LIN {X 0,Y 566.531,Z 316.319,A -85,B 0,C 180,E1 -2651.108,E2 -2651.108} C_VEL
LIN {X 0,Y 566.471,Z 313.294,A -85,B 0,C 180,E1 -2653.028,E2 -2653.028} C_VEL
LIN {X 0,Y 566.256,Z 311.81,A -85,B 0,C 180,E1 -2654.03,E2 -2654.03} C_VEL
LIN {X 0,Y 566.196,Z 311.46,A -85,B 0,C 180,E1 -2656.049,E2 -2656.049} C_VEL
LIN {X 0,Y 566.205,Z 311.453,A -85,B 0,C 180,E1 -2659.214,E2 -2659.214} C_VEL
LIN {X 0,Y 566.187,Z 311.457,A -85,B 0,C 180,E1 -2661.637,E2 -2661.637} C_VEL
LIN {X 0,Y 566.162,Z 311.463,A -85,B 0,C 180,E1 -2664.308,E2 -2664.308} C_VEL
LIN {X 0,Y 566.22,Z 311.449,A -85,B 0,C 180,E1 -2666.897,E2 -2666.897} C_VEL
LIN {X 0,Y 566.18,Z 311.456,A -85,B 0,C 180,E1 -2669.407,E2 -2669.407} C_VEL
LIN {X 0,Y 566.212,Z 311.46,A -85,B 0,C 180,E1 -2671.857,E2 -2671.857} C_VEL
LIN {X 0,Y 566.214,Z 311.452,A -85,B 0,C 180,E1 -2674.251,E2 -2674.251} C_VEL
LIN {X 0,Y 566.169,Z 311.455,A -85,B 0,C 180,E1 -2676.719,E2 -2676.719} C_VEL
LIN {X 0,Y 566.207,Z 311.46,A -85,B 0,C 180,E1 -2679.662,E2 -2679.662} C_VEL
LIN {X 0,Y 566.198,Z 311.451,A -85,B 0,C 180,E1 -2682.668,E2 -2682.668} C_VEL
LIN {X 0,Y 566.234,Z 311.455,A -85,B 0,C 180,E1 -2685.626,E2 -2685.626} C_VEL
LIN {X 0,Y 566.235,Z 311.447,A -85,B 0,C 180,E1 -2688.675,E2 -2688.675} C_VEL
LIN {X 0,Y 566.233,Z 311.456,A -85,B 0,C 180,E1 -2691.434,E2 -2691.434} C_VEL
LIN {X 0,Y 566.262,Z 311.443,A -85,B 0,C 180,E1 -2694.301,E2 -2694.301} C_VEL
LIN {X 0,Y 566.286,Z 311.442,A -85,B 0,C 180,E1 -2697.866,E2 -2697.866} C_VEL
LIN {X 0,Y 566.297,Z 311.442,A -85,B 0,C 180,E1 -2700.711,E2 -2700.711} C_VEL
LIN {X 0,Y 566.268,Z 311.448,A -85,B 0,C 180,E1 -2702.845,E2 -2702.845} C_VEL
LIN {X 0,Y 566.266,Z 311.444,A -85,B 0,C 180,E1 -2705.698,E2 -2705.698} C_VEL
LIN {X 0,Y 566.226,Z 311.452,A -85,B 0,C 180,E1 -2708.565,E2 -2708.565} C_VEL
LIN {X 0,Y 566.241,Z 311.448,A -85,B 0,C 180,E1 -2711.454,E2 -2711.454} C_VEL
LIN {X 0,Y 566.233,Z 311.452,A -85,B 0,C 180,E1 -2714.506,E2 -2714.506} C_VEL
LIN {X 0,Y 566.197,Z 311.453,A -85,B 0,C 180,E1 -2717.331,E2 -2717.331} C_VEL
LIN {X 0,Y 566.211,Z 311.454,A -85,B 0,C 180,E1 -2720.337,E2 -2720.337} C_VEL
LIN {X 0,Y 566.17,Z 311.456,A -85,B 0,C 180,E1 -2723.281,E2 -2723.281} C_VEL
LIN {X 0,Y 566.212,Z 311.45,A -85,B 0,C 180,E1 -2725.749,E2 -2725.749} C_VEL
LIN {X 0,Y 566.201,Z 311.451,A -85,B 0,C 180,E1 -2727.472,E2 -2727.472} C_VEL
LIN {X 0,Y 565.52,Z 311.541,A -85,B 0,C 180,E1 -2728.066,E2 -2728.066} C_VEL
LIN {X 0,Y 562.655,Z 311.896,A -85,B 0,C 180,E1 -2729.029,E2 -2729.029} C_VEL
LIN {X 0,Y 560.247,Z 312.196,A -85,B 0,C 180,E1 -2729.805,E2 -2729.805} C_VEL
LIN {X 0,Y 559.222,Z 312.33,A -85,B 0,C 180,E1 -2730.404,E2 -2730.404} C_VEL
LIN {X 0,Y 559.142,Z 312.332,A -85,B 0,C 180,E1 -2730.606,E2 -2730.606} C_VEL
LIN {X 0,Y 559.173,Z 312.331,A -85,B 0,C 180,E1 -2732.714,E2 -2732.714} C_VEL
LIN {X 0,Y 559.141,Z 312.33,A -85,B 0,C 180,E1 -2735.323,E2 -2735.323} C_VEL
LIN {X 0,Y 559.133,Z 312.337,A -85,B 0,C 180,E1 -2738.017,E2 -2738.017} C_VEL
LIN {X 0,Y 559.173,Z 312.328,A -85,B 0,C 180,E1 -2740.81,E2 -2740.81} C_VEL
LIN {X 0,Y 559.16,Z 312.332,A -85,B 0,C 180,E1 -2743.731,E2 -2743.731} C_VEL
LIN {X 0,Y 559.146,Z 312.33,A -85,B 0,C 180,E1 -2746.803,E2 -2746.803} C_VEL
LIN {X 0,Y 559.173,Z 312.327,A -85,B 0,C 180,E1 -2749.189,E2 -2749.189} C_VEL
LIN {X 0,Y 559.132,Z 312.34,A -85,B 0,C 180,E1 -2751.983,E2 -2751.983} C_VEL
LIN {X 0,Y 559.143,Z 312.33,A -85,B 0,C 180,E1 -2754.785,E2 -2754.785} C_VEL
LIN {X 0,Y 559.171,Z 312.33,A -85,B 0,C 180,E1 -2757.361,E2 -2757.361} C_VEL
LIN {X 0,Y 559.146,Z 312.333,A -85,B 0,C 180,E1 -2760.142,E2 -2760.142} C_VEL
LIN {X 0,Y 559.179,Z 312.328,A -85,B 0,C 180,E1 -2763.17,E2 -2763.17} C_VEL
LIN {X 0,Y 559.154,Z 312.337,A -85,B 0,C 180,E1 -2765.495,E2 -2765.495} C_VEL
LIN {X 0,Y 559.169,Z 312.327,A -85,B 0,C 180,E1 -2768.624,E2 -2768.624} C_VEL
LIN {X 0,Y 559.166,Z 312.33,A -85,B 0,C 180,E1 -2770.926,E2 -2770.926} C_VEL
LIN {X 0,Y 559.164,Z 312.331,A -85,B 0,C 180,E1 -2773.948,E2 -2773.948} C_VEL
LIN {X 0,Y 559.169,Z 312.328,A -85,B 0,C 180,E1 -2776.184,E2 -2776.184} C_VEL
LIN {X 0,Y 559.194,Z 312.332,A -85,B 0,C 180,E1 -2779.134,E2 -2779.134} C_VEL
LIN {X 0,Y 559.203,Z 312.324,A -85,B 0,C 180,E1 -2782.054,E2 -2782.054} C_VEL
LIN {X 0,Y 559.253,Z 312.325,A -85,B 0,C 180,E1 -2784.953,E2 -2784.953} C_VEL
LIN {X 0,Y 559.255,Z 312.318,A -85,B 0,C 180,E1 -2787.839,E2 -2787.839} C_VEL
LIN {X 0,Y 559.27,Z 312.321,A -85,B 0,C 180,E1 -2790.72,E2 -2790.72} C_VEL
LIN {X 0,Y 559.236,Z 312.328,A -85,B 0,C 180,E1 -2792.881,E2 -2792.881} C_VEL
LIN {X 0,Y 559.235,Z 312.32,A -85,B 0,C 180,E1 -2795.77,E2 -2795.77} C_VEL
LIN {X 0,Y 559.189,Z 312.333,A -85,B 0,C 180,E1 -2798.674,E2 -2798.674} C_VEL
LIN {X 0,Y 559.202,Z 312.324,A -85,B 0,C 180,E1 -2801.6,E2 -2801.6} C_VEL
LIN {X 0,Y 559.197,Z 312.333,A -85,B 0,C 180,E1 -2804.596,E2 -2804.596} C_VEL
LIN {X 0,Y 559.157,Z 312.33,A -85,B 0,C 180,E1 -2807.557,E2 -2807.557} C_VEL
LIN {X 0,Y 559.17,Z 312.328,A -85,B 0,C 180,E1 -2809.837,E2 -2809.837} C_VEL
LIN {X 0,Y 559.139,Z 312.336,A -85,B 0,C 180,E1 -2812.153,E2 -2812.153} C_VEL
LIN {X 0,Y 559.175,Z 312.326,A -85,B 0,C 180,E1 -2815.298,E2 -2815.298} C_VEL
LIN {X 0,Y 559.192,Z 312.326,A -85,B 0,C 180,E1 -2817.711,E2 -2817.711} C_VEL
LIN {X 0,Y 559.16,Z 312.329,A -85,B 0,C 180,E1 -2821.019,E2 -2821.019} C_VEL
LIN {X 0,Y 559.162,Z 312.334,A -85,B 0,C 180,E1 -2823.949,E2 -2823.949} C_VEL
LIN {X 0,Y 559.142,Z 312.33,A -85,B 0,C 180,E1 -2827.108,E2 -2827.108} C_VEL
LIN {X 0,Y 559.167,Z 312.336,A -85,B 0,C 180,E1 -2829.943,E2 -2829.943} C_VEL
LIN {X 0,Y 559.16,Z 312.329,A -85,B 0,C 180,E1 -2832.743,E2 -2832.743} C_VEL
LIN {X 0,Y 559.152,Z 312.337,A -85,B 0,C 180,E1 -2835.761,E2 -2835.761} C_VEL
LIN {X 0,Y 559.189,Z 312.328,A -85,B 0,C 180,E1 -2838.233,E2 -2838.233} C_VEL
LIN {X 0,Y 559.175,Z 312.328,A -85,B 0,C 180,E1 -2841.191,E2 -2841.191} C_VEL
LIN {X 0,Y 559.136,Z 312.339,A -85,B 0,C 180,E1 -2843.79,E2 -2843.79} C_VEL
LIN {X 0,Y 559.162,Z 312.328,A -85,B 0,C 180,E1 -2846.426,E2 -2846.426} C_VEL
LIN {X 0,Y 559.16,Z 312.33,A -85,B 0,C 180,E1 -2848.982,E2 -2848.982} C_VEL
LIN {X 0,Y 559.165,Z 312.335,A -85,B 0,C 180,E1 -2851.619,E2 -2851.619} C_VEL
LIN {X 0,Y 559.179,Z 312.329,A -85,B 0,C 180,E1 -2853.903,E2 -2853.903} C_VEL
LIN {X 0,Y 559.14,Z 312.331,A -85,B 0,C 180,E1 -2856.571,E2 -2856.571} C_VEL
LIN {X 0,Y 559.178,Z 312.335,A -85,B 0,C 180,E1 -2859.396,E2 -2859.396} C_VEL
LIN {X 0,Y 559.144,Z 312.333,A -85,B 0,C 180,E1 -2861.686,E2 -2861.686} C_VEL
LIN {X 0,Y 559.163,Z 312.328,A -85,B 0,C 180,E1 -2863.948,E2 -2863.948} C_VEL
LIN {X 0,Y 559.17,Z 312.327,A -85,B 0,C 180,E1 -2866.184,E2 -2866.184} C_VEL
LIN {X 0,Y 559.194,Z 312.333,A -85,B 0,C 180,E1 -2869.134,E2 -2869.134} C_VEL
LIN {X 0,Y 559.202,Z 312.323,A -85,B 0,C 180,E1 -2872.054,E2 -2872.054} C_VEL
LIN {X 0,Y 559.252,Z 312.327,A -85,B 0,C 180,E1 -2874.954,E2 -2874.954} C_VEL
LIN {X 0,Y 559.255,Z 312.316,A -85,B 0,C 180,E1 -2877.84,E2 -2877.84} C_VEL
LIN {X 0,Y 559.274,Z 312.322,A -85,B 0,C 180,E1 -2880.72,E2 -2880.72} C_VEL
LIN {X 0,Y 559.237,Z 312.326,A -85,B 0,C 180,E1 -2882.882,E2 -2882.882} C_VEL
LIN {X 0,Y 559.231,Z 312.319,A -85,B 0,C 180,E1 -2885.771,E2 -2885.771} C_VEL
LIN {X 0,Y 559.191,Z 312.333,A -85,B 0,C 180,E1 -2888.675,E2 -2888.675} C_VEL
LIN {X 0,Y 559.205,Z 312.323,A -85,B 0,C 180,E1 -2891.601,E2 -2891.601} C_VEL
LIN {X 0,Y 559.2,Z 312.331,A -85,B 0,C 180,E1 -2894.596,E2 -2894.596} C_VEL
LIN {X 0,Y 559.142,Z 312.331,A -85,B 0,C 180,E1 -2897.558,E2 -2897.558} C_VEL
LIN {X 0,Y 559.166,Z 312.33,A -85,B 0,C 180,E1 -2899.838,E2 -2899.838} C_VEL
LIN {X 0,Y 559.142,Z 312.338,A -85,B 0,C 180,E1 -2902.153,E2 -2902.153} C_VEL
LIN {X 0,Y 559.176,Z 312.326,A -85,B 0,C 180,E1 -2905.298,E2 -2905.298} C_VEL
LIN {X 0,Y 559.157,Z 312.332,A -85,B 0,C 180,E1 -2907.714,E2 -2907.714} C_VEL
LIN {X 0,Y 559.153,Z 312.337,A -85,B 0,C 180,E1 -2910.183,E2 -2910.183} C_VEL
LIN {X 0,Y 559.157,Z 312.329,A -85,B 0,C 180,E1 -2912.716,E2 -2912.716} C_VEL
LIN {X 0,Y 559.127,Z 312.333,A -85,B 0,C 180,E1 -2915.324,E2 -2915.324} C_VEL
LIN {X 0,Y 559.134,Z 312.341,A -85,B 0,C 180,E1 -2918.018,E2 -2918.018} C_VEL
LIN {X 0,Y 559.156,Z 312.331,A -85,B 0,C 180,E1 -2920.813,E2 -2920.813} C_VEL
LIN {X 0,Y 559.14,Z 312.34,A -85,B 0,C 180,E1 -2923.734,E2 -2923.734} C_VEL
LIN {X 0,Y 559.151,Z 312.338,A -85,B 0,C 180,E1 -2925.262,E2 -2925.262} C_VEL
LIN {X 0,Y 559.431,Z 314.242,A -85,B 0,C 180,E1 -2926.773,E2 -2926.773} C_VEL
LIN {X 0,Y 559.539,Z 318.057,A -85,B 0,C 180,E1 -2929.222,E2 -2929.222} C_VEL
LIN {X 0,Y 559.468,Z 322.75,A -85,B 0,C 180,E1 -2932.009,E2 -2932.009} C_VEL
LIN {X 0,Y 559.387,Z 327.696,A -85,B 0,C 180,E1 -2934.751,E2 -2934.751} C_VEL
LIN {X 0,Y 559.313,Z 332.663,A -85,B 0,C 180,E1 -2937.34,E2 -2937.34} C_VEL
LIN {X 0,Y 559.203,Z 338.301,A -85,B 0,C 180,E1 -2940.134,E2 -2940.134} C_VEL
LIN {X 0,Y 559.094,Z 344.792,A -85,B 0,C 180,E1 -2943.189,E2 -2943.189} C_VEL
LIN {X 0,Y 559.019,Z 349.846,A -85,B 0,C 180,E1 -2945.489,E2 -2945.489} C_VEL
LIN {X 0,Y 558.987,Z 357.018,A -85,B 0,C 180,E1 -2948.617,E2 -2948.617} C_VEL
LIN {X 0,Y 558.928,Z 362.478,A -85,B 0,C 180,E1 -2950.918,E2 -2950.918} C_VEL
LIN {X 0,Y 558.876,Z 367.867,A -85,B 0,C 180,E1 -2953.188,E2 -2953.188} C_VEL
LIN {X 0,Y 558.841,Z 375.053,A -85,B 0,C 180,E1 -2956.176,E2 -2956.176} C_VEL
LIN {X 0,Y 558.832,Z 377.523,A -85,B 0,C 180,E1 -2957.194,E2 -2957.194} C_VEL
LIN {X 0,Y 559.957,Z 385.372,A -85,B 0,C 180,E1 -2957.381,E2 -2957.381} C_VEL
LIN {X 0,Y 559.843,Z 397.181,A -85,B 0,C 180,E1 -2957.728,E2 -2957.728} C_VEL
LIN {X 0,Y 559.719,Z 408.183,A -85,B 0,C 180,E1 -2958.171,E2 -2958.171} C_VEL
LIN {X 0,Y 559.565,Z 418.532,A -85,B 0,C 180,E1 -2958.704,E2 -2958.704} C_VEL
LIN {X 0,Y 559.421,Z 429.49,A -85,B 0,C 180,E1 -2959.413,E2 -2959.413} C_VEL
LIN {X 0,Y 559.289,Z 439.624,A -85,B 0,C 180,E1 -2960.233,E2 -2960.233} C_VEL
LIN {X 0,Y 559.138,Z 448.736,A -85,B 0,C 180,E1 -2961.143,E2 -2961.143} C_VEL
LIN {X 0,Y 559.052,Z 456.283,A -85,B 0,C 180,E1 -2962.051,E2 -2962.051} C_VEL
LIN {X 0,Y 558.934,Z 462.688,A -85,B 0,C 180,E1 -2962.976,E2 -2962.976} C_VEL
LIN {X 0,Y 558.908,Z 467.807,A -85,B 0,C 180,E1 -2963.864,E2 -2963.864} C_VEL
LIN {X 0,Y 558.798,Z 472.904,A -85,B 0,C 180,E1 -2964.949,E2 -2964.949} C_VEL
LIN {X 0,Y 558.844,Z 476.858,A -85,B 0,C 180,E1 -2966.034,E2 -2966.034} C_VEL
LIN {X 0,Y 558.799,Z 479.778,A -85,B 0,C 180,E1 -2967.116,E2 -2967.116} C_VEL
LIN {X 0,Y 558.745,Z 482.194,A -85,B 0,C 180,E1 -2968.559,E2 -2968.559} C_VEL
LIN {X 0,Y 558.741,Z 482.781,A -85,B 0,C 180,E1 -2969.279,E2 -2969.279} C_VEL
LIN {X 0,Y 558.741,Z 482.781,A -85,B 0,C 180,E1 -2970.721,E2 -2970.721} C_VEL
LIN {X 0,Y 558.745,Z 482.194,A -85,B 0,C 180,E1 -2971.441,E2 -2971.441} C_VEL
LIN {X 0,Y 558.799,Z 479.778,A -85,B 0,C 180,E1 -2972.884,E2 -2972.884} C_VEL
LIN {X 0,Y 558.844,Z 476.858,A -85,B 0,C 180,E1 -2973.966,E2 -2973.966} C_VEL
LIN {X 0,Y 558.798,Z 472.904,A -85,B 0,C 180,E1 -2975.051,E2 -2975.051} C_VEL
LIN {X 0,Y 558.91,Z 467.807,A -85,B 0,C 180,E1 -2976.136,E2 -2976.136} C_VEL
LIN {X 0,Y 558.975,Z 461.423,A -85,B 0,C 180,E1 -2977.223,E2 -2977.223} C_VEL
LIN {X 0,Y 559.093,Z 453.5,A -85,B 0,C 180,E1 -2978.312,E2 -2978.312} C_VEL
LIN {X 0,Y 559.21,Z 445.358,A -85,B 0,C 180,E1 -2979.221,E2 -2979.221} C_VEL
LIN {X 0,Y 559.345,Z 435.315,A -85,B 0,C 180,E1 -2980.131,E2 -2980.131} C_VEL
LIN {X 0,Y 559.473,Z 426.835,A -85,B 0,C 180,E1 -2980.769,E2 -2980.769} C_VEL
LIN {X 0,Y 559.575,Z 416.58,A -85,B 0,C 180,E1 -2981.405,E2 -2981.405} C_VEL
LIN {X 0,Y 559.736,Z 405.396,A -85,B 0,C 180,E1 -2981.956,E2 -2981.956} C_VEL
LIN {X 0,Y 559.931,Z 392.286,A -85,B 0,C 180,E1 -2982.435,E2 -2982.435} C_VEL
LIN {X 0,Y 559.761,Z 383.139,A -85,B 0,C 180,E1 -2982.678,E2 -2982.678} C_VEL
LIN {X 0,Y 558.832,Z 377.523,A -85,B 0,C 180,E1 -2982.806,E2 -2982.806} C_VEL
LIN {X 0,Y 558.852,Z 371.46,A -85,B 0,C 180,E1 -2985.313,E2 -2985.313} C_VEL
LIN {X 0,Y 558.903,Z 364.274,A -85,B 0,C 180,E1 -2988.322,E2 -2988.322} C_VEL
LIN {X 0,Y 558.932,Z 358.847,A -85,B 0,C 180,E1 -2990.614,E2 -2990.614} C_VEL
LIN {X 0,Y 558.97,Z 352.352,A -85,B 0,C 180,E1 -2993.387,E2 -2993.387} C_VEL
LIN {X 0,Y 559.064,Z 346.339,A -85,B 0,C 180,E1 -2996.103,E2 -2996.103} C_VEL
LIN {X 0,Y 559.116,Z 341.086,A -85,B 0,C 180,E1 -2998.532,E2 -2998.532} C_VEL
LIN {X 0,Y 559.232,Z 335.376,A -85,B 0,C 180,E1 -3001.287,E2 -3001.287} C_VEL
LIN {X 0,Y 559.298,Z 330.113,A -85,B 0,C 180,E1 -3003.969,E2 -3003.969} C_VEL
LIN {X 0,Y 559.418,Z 325.417,A -85,B 0,C 180,E1 -3006.482,E2 -3006.482} C_VEL
LIN {X 0,Y 559.507,Z 321.151,A -85,B 0,C 180,E1 -3008.906,E2 -3008.906} C_VEL
LIN {X 0,Y 559.54,Z 316.507,A -85,B 0,C 180,E1 -3011.736,E2 -3011.736} C_VEL
LIN {X 0,Y 559.319,Z 313.521,A -85,B 0,C 180,E1 -3013.716,E2 -3013.716} C_VEL
LIN {X 0,Y 559.151,Z 312.337,A -85,B 0,C 180,E1 -3014.738,E2 -3014.738} C_VEL
LIN {X 0,Y 559.156,Z 312.336,A -85,B 0,C 180,E1 -3017.865,E2 -3017.865} C_VEL
LIN {X 0,Y 559.185,Z 312.335,A -85,B 0,C 180,E1 -3020.134,E2 -3020.134} C_VEL
LIN {X 0,Y 559.141,Z 312.332,A -85,B 0,C 180,E1 -3022.891,E2 -3022.891} C_VEL
LIN {X 0,Y 559.166,Z 312.336,A -85,B 0,C 180,E1 -3026.051,E2 -3026.051} C_VEL
LIN {X 0,Y 559.155,Z 312.329,A -85,B 0,C 180,E1 -3028.98,E2 -3028.98} C_VEL
LIN {X 0,Y 559.169,Z 312.333,A -85,B 0,C 180,E1 -3031.618,E2 -3031.618} C_VEL
LIN {X 0,Y 559.18,Z 312.334,A -85,B 0,C 180,E1 -3033.903,E2 -3033.903} C_VEL
LIN {X 0,Y 559.139,Z 312.331,A -85,B 0,C 180,E1 -3036.571,E2 -3036.571} C_VEL
LIN {X 0,Y 559.176,Z 312.331,A -85,B 0,C 180,E1 -3039.395,E2 -3039.395} C_VEL
LIN {X 0,Y 559.142,Z 312.339,A -85,B 0,C 180,E1 -3041.685,E2 -3041.685} C_VEL
LIN {X 0,Y 559.166,Z 312.331,A -85,B 0,C 180,E1 -3043.947,E2 -3043.947} C_VEL
LIN {X 0,Y 559.17,Z 312.328,A -85,B 0,C 180,E1 -3046.184,E2 -3046.184} C_VEL
LIN {X 0,Y 559.196,Z 312.328,A -85,B 0,C 180,E1 -3049.133,E2 -3049.133} C_VEL
LIN {X 0,Y 559.201,Z 312.324,A -85,B 0,C 180,E1 -3052.053,E2 -3052.053} C_VEL
LIN {X 0,Y 559.254,Z 312.321,A -85,B 0,C 180,E1 -3054.953,E2 -3054.953} C_VEL
LIN {X 0,Y 559.256,Z 312.318,A -85,B 0,C 180,E1 -3057.839,E2 -3057.839} C_VEL
LIN {X 0,Y 559.268,Z 312.318,A -85,B 0,C 180,E1 -3060.72,E2 -3060.72} C_VEL
LIN {X 0,Y 559.235,Z 312.325,A -85,B 0,C 180,E1 -3062.881,E2 -3062.881} C_VEL
LIN {X 0,Y 559.234,Z 312.32,A -85,B 0,C 180,E1 -3065.77,E2 -3065.77} C_VEL
LIN {X 0,Y 559.185,Z 312.33,A -85,B 0,C 180,E1 -3068.674,E2 -3068.674} C_VEL
LIN {X 0,Y 559.204,Z 312.324,A -85,B 0,C 180,E1 -3071.6,E2 -3071.6} C_VEL
LIN {X 0,Y 559.198,Z 312.329,A -85,B 0,C 180,E1 -3074.595,E2 -3074.595} C_VEL
LIN {X 0,Y 559.157,Z 312.329,A -85,B 0,C 180,E1 -3077.557,E2 -3077.557} C_VEL
LIN {X 0,Y 559.17,Z 312.327,A -85,B 0,C 180,E1 -3079.837,E2 -3079.837} C_VEL
LIN {X 0,Y 559.14,Z 312.333,A -85,B 0,C 180,E1 -3082.152,E2 -3082.152} C_VEL
LIN {X 0,Y 559.173,Z 312.327,A -85,B 0,C 180,E1 -3085.298,E2 -3085.298} C_VEL
LIN {X 0,Y 559.178,Z 312.326,A -85,B 0,C 180,E1 -3087.712,E2 -3087.712} C_VEL
LIN {X 0,Y 559.142,Z 312.332,A -85,B 0,C 180,E1 -3090.606,E2 -3090.606} C_VEL
LIN {X 0,Y 558.482,Z 312.415,A -85,B 0,C 180,E1 -3091.208,E2 -3091.208} C_VEL
LIN {X 0,Y 555.622,Z 312.775,A -85,B 0,C 180,E1 -3092.184,E2 -3092.184} C_VEL
LIN {X 0,Y 553.208,Z 313.072,A -85,B 0,C 180,E1 -3092.97,E2 -3092.97} C_VEL
LIN {X 0,Y 552.185,Z 313.198,A -85,B 0,C 180,E1 -3093.576,E2 -3093.576} C_VEL
LIN {X 0,Y 552.11,Z 313.208,A -85,B 0,C 180,E1 -3093.782,E2 -3093.782} C_VEL
LIN {X 0,Y 552.106,Z 313.21,A -85,B 0,C 180,E1 -3096.746,E2 -3096.746} C_VEL
LIN {X 0,Y 552.131,Z 313.205,A -85,B 0,C 180,E1 -3099.526,E2 -3099.526} C_VEL
LIN {X 0,Y 552.127,Z 313.209,A -85,B 0,C 180,E1 -3102.425,E2 -3102.425} C_VEL
LIN {X 0,Y 552.096,Z 313.21,A -85,B 0,C 180,E1 -3105.563,E2 -3105.563} C_VEL
LIN {X 0,Y 552.137,Z 313.204,A -85,B 0,C 180,E1 -3108.676,E2 -3108.676} C_VEL
LIN {X 0,Y 552.117,Z 313.208,A -85,B 0,C 180,E1 -3111.411,E2 -3111.411} C_VEL
LIN {X 0,Y 552.099,Z 313.213,A -85,B 0,C 180,E1 -3114.158,E2 -3114.158} C_VEL
LIN {X 0,Y 552.12,Z 313.205,A -85,B 0,C 180,E1 -3116.815,E2 -3116.815} C_VEL
LIN {X 0,Y 552.104,Z 313.211,A -85,B 0,C 180,E1 -3119.391,E2 -3119.391} C_VEL
LIN {X 0,Y 552.124,Z 313.211,A -85,B 0,C 180,E1 -3121.903,E2 -3121.903} C_VEL
LIN {X 0,Y 552.154,Z 313.201,A -85,B 0,C 180,E1 -3124.649,E2 -3124.649} C_VEL
LIN {X 0,Y 552.09,Z 313.219,A -85,B 0,C 180,E1 -3127.549,E2 -3127.549} C_VEL
LIN {X 0,Y 552.146,Z 313.202,A -85,B 0,C 180,E1 -3130.373,E2 -3130.373} C_VEL
LIN {X 0,Y 552.152,Z 313.205,A -85,B 0,C 180,E1 -3132.977,E2 -3132.977} C_VEL
LIN {X 0,Y 552.133,Z 313.206,A -85,B 0,C 180,E1 -3136.004,E2 -3136.004} C_VEL
LIN {X 0,Y 552.161,Z 313.206,A -85,B 0,C 180,E1 -3138.993,E2 -3138.993} C_VEL
LIN {X 0,Y 552.157,Z 313.203,A -85,B 0,C 180,E1 -3141.952,E2 -3141.952} C_VEL
LIN {X 0,Y 552.228,Z 313.199,A -85,B 0,C 180,E1 -3144.889,E2 -3144.889} C_VEL
LIN {X 0,Y 552.225,Z 313.194,A -85,B 0,C 180,E1 -3147.812,E2 -3147.812} C_VEL
LIN {X 0,Y 552.24,Z 313.197,A -85,B 0,C 180,E1 -3150.729,E2 -3150.729} C_VEL
LIN {X 0,Y 552.202,Z 313.204,A -85,B 0,C 180,E1 -3152.918,E2 -3152.918} C_VEL
LIN {X 0,Y 552.205,Z 313.196,A -85,B 0,C 180,E1 -3155.844,E2 -3155.844} C_VEL
LIN {X 0,Y 552.16,Z 313.21,A -85,B 0,C 180,E1 -3158.786,E2 -3158.786} C_VEL
LIN {X 0,Y 552.16,Z 313.201,A -85,B 0,C 180,E1 -3161.75,E2 -3161.75} C_VEL
LIN {X 0,Y 552.133,Z 313.213,A -85,B 0,C 180,E1 -3164.748,E2 -3164.748} C_VEL
LIN {X 0,Y 552.108,Z 313.208,A -85,B 0,C 180,E1 -3167.788,E2 -3167.788} C_VEL
LIN {X 0,Y 552.128,Z 313.208,A -85,B 0,C 180,E1 -3170.101,E2 -3170.101} C_VEL
LIN {X 0,Y 552.09,Z 313.219,A -85,B 0,C 180,E1 -3172.451,E2 -3172.451} C_VEL
LIN {X 0,Y 552.154,Z 313.201,A -85,B 0,C 180,E1 -3175.351,E2 -3175.351} C_VEL
LIN {X 0,Y 552.124,Z 313.211,A -85,B 0,C 180,E1 -3178.097,E2 -3178.097} C_VEL
LIN {X 0,Y 552.104,Z 313.211,A -85,B 0,C 180,E1 -3180.609,E2 -3180.609} C_VEL
LIN {X 0,Y 552.12,Z 313.205,A -85,B 0,C 180,E1 -3183.185,E2 -3183.185} C_VEL
LIN {X 0,Y 552.099,Z 313.213,A -85,B 0,C 180,E1 -3185.842,E2 -3185.842} C_VEL
LIN {X 0,Y 552.123,Z 313.205,A -85,B 0,C 180,E1 -3189.062,E2 -3189.062} C_VEL
LIN {X 0,Y 552.137,Z 313.205,A -85,B 0,C 180,E1 -3191.444,E2 -3191.444} C_VEL
LIN {X 0,Y 552.093,Z 313.21,A -85,B 0,C 180,E1 -3194.532,E2 -3194.532} C_VEL
LIN {X 0,Y 552.128,Z 313.21,A -85,B 0,C 180,E1 -3197.585,E2 -3197.585} C_VEL
LIN {X 0,Y 552.131,Z 313.205,A -85,B 0,C 180,E1 -3200.474,E2 -3200.474} C_VEL
LIN {X 0,Y 552.103,Z 313.211,A -85,B 0,C 180,E1 -3203.317,E2 -3203.317} C_VEL
LIN {X 0,Y 552.124,Z 313.21,A -85,B 0,C 180,E1 -3205.939,E2 -3205.939} C_VEL
LIN {X 0,Y 552.116,Z 313.206,A -85,B 0,C 180,E1 -3208.541,E2 -3208.541} C_VEL
LIN {X 0,Y 552.122,Z 313.213,A -85,B 0,C 180,E1 -3211.438,E2 -3211.438} C_VEL
LIN {X 0,Y 552.128,Z 313.204,A -85,B 0,C 180,E1 -3214.356,E2 -3214.356} C_VEL
LIN {X 0,Y 552.097,Z 313.209,A -85,B 0,C 180,E1 -3216.758,E2 -3216.758} C_VEL
LIN {X 0,Y 552.119,Z 313.212,A -85,B 0,C 180,E1 -3219.12,E2 -3219.12} C_VEL
LIN {X 0,Y 552.123,Z 313.211,A -85,B 0,C 180,E1 -3221.445,E2 -3221.445} C_VEL
LIN {X 0,Y 552.113,Z 313.208,A -85,B 0,C 180,E1 -3223.738,E2 -3223.738} C_VEL
LIN {X 0,Y 552.134,Z 313.204,A -85,B 0,C 180,E1 -3226.005,E2 -3226.005} C_VEL
LIN {X 0,Y 552.161,Z 313.208,A -85,B 0,C 180,E1 -3228.994,E2 -3228.994} C_VEL
LIN {X 0,Y 552.156,Z 313.201,A -85,B 0,C 180,E1 -3231.952,E2 -3231.952} C_VEL
LIN {X 0,Y 552.227,Z 313.201,A -85,B 0,C 180,E1 -3234.889,E2 -3234.889} C_VEL
LIN {X 0,Y 552.226,Z 313.192,A -85,B 0,C 180,E1 -3237.812,E2 -3237.812} C_VEL
LIN {X 0,Y 552.244,Z 313.198,A -85,B 0,C 180,E1 -3240.73,E2 -3240.73} C_VEL
LIN {X 0,Y 552.203,Z 313.202,A -85,B 0,C 180,E1 -3242.919,E2 -3242.919} C_VEL
LIN {X 0,Y 552.201,Z 313.195,A -85,B 0,C 180,E1 -3245.844,E2 -3245.844} C_VEL
LIN {X 0,Y 552.162,Z 313.207,A -85,B 0,C 180,E1 -3248.786,E2 -3248.786} C_VEL
LIN {X 0,Y 552.162,Z 313.2,A -85,B 0,C 180,E1 -3251.751,E2 -3251.751} C_VEL
LIN {X 0,Y 552.136,Z 313.208,A -85,B 0,C 180,E1 -3254.749,E2 -3254.749} C_VEL
LIN {X 0,Y 552.1,Z 313.209,A -85,B 0,C 180,E1 -3257.789,E2 -3257.789} C_VEL
LIN {X 0,Y 552.127,Z 313.21,A -85,B 0,C 180,E1 -3260.102,E2 -3260.102} C_VEL
LIN {X 0,Y 552.092,Z 313.215,A -85,B 0,C 180,E1 -3262.451,E2 -3262.451} C_VEL
LIN {X 0,Y 552.156,Z 313.201,A -85,B 0,C 180,E1 -3265.351,E2 -3265.351} C_VEL
LIN {X 0,Y 552.11,Z 313.215,A -85,B 0,C 180,E1 -3268.099,E2 -3268.099} C_VEL
LIN {X 0,Y 552.102,Z 313.21,A -85,B 0,C 180,E1 -3270.61,E2 -3270.61} C_VEL
LIN {X 0,Y 552.116,Z 313.206,A -85,B 0,C 180,E1 -3273.186,E2 -3273.186} C_VEL
LIN {X 0,Y 552.086,Z 313.217,A -85,B 0,C 180,E1 -3275.844,E2 -3275.844} C_VEL
LIN {X 0,Y 552.125,Z 313.207,A -85,B 0,C 180,E1 -3279.062,E2 -3279.062} C_VEL
LIN {X 0,Y 552.122,Z 313.212,A -85,B 0,C 180,E1 -3281.446,E2 -3281.446} C_VEL
LIN {X 0,Y 552.095,Z 313.215,A -85,B 0,C 180,E1 -3284.532,E2 -3284.532} C_VEL
LIN {X 0,Y 552.171,Z 313.752,A -85,B 0,C 180,E1 -3285.57,E2 -3285.57} C_VEL
LIN {X 0,Y 552.532,Z 316.734,A -85,B 0,C 180,E1 -3287.613,E2 -3287.613} C_VEL
LIN {X 0,Y 552.491,Z 321.334,A -85,B 0,C 180,E1 -3290.504,E2 -3290.504} C_VEL
LIN {X 0,Y 552.436,Z 326.103,A -85,B 0,C 180,E1 -3293.279,E2 -3293.279} C_VEL
LIN {X 0,Y 552.298,Z 330.997,A -85,B 0,C 180,E1 -3295.951,E2 -3295.951} C_VEL
LIN {X 0,Y 552.203,Z 336.005,A -85,B 0,C 180,E1 -3298.546,E2 -3298.546} C_VEL
LIN {X 0,Y 552.084,Z 341.909,A -85,B 0,C 180,E1 -3301.446,E2 -3301.446} C_VEL
LIN {X 0,Y 551.994,Z 348.09,A -85,B 0,C 180,E1 -3304.349,E2 -3304.349} C_VEL
LIN {X 0,Y 551.88,Z 355.104,A -85,B 0,C 180,E1 -3307.54,E2 -3307.54} C_VEL
LIN {X 0,Y 551.884,Z 361.908,A -85,B 0,C 180,E1 -3310.452,E2 -3310.452} C_VEL
LIN {X 0,Y 551.816,Z 367.867,A -85,B 0,C 180,E1 -3312.967,E2 -3312.967} C_VEL
LIN {X 0,Y 551.755,Z 375.053,A -85,B 0,C 180,E1 -3315.995,E2 -3315.995} C_VEL
LIN {X 0,Y 551.73,Z 377.523,A -85,B 0,C 180,E1 -3317.026,E2 -3317.026} C_VEL
LIN {X 0,Y 553.023,Z 386.217,A -85,B 0,C 180,E1 -3317.244,E2 -3317.244} C_VEL
LIN {X 0,Y 552.921,Z 397.035,A -85,B 0,C 180,E1 -3317.568,E2 -3317.568} C_VEL
LIN {X 0,Y 552.772,Z 407.382,A -85,B 0,C 180,E1 -3317.984,E2 -3317.984} C_VEL
LIN {X 0,Y 552.622,Z 417.171,A -85,B 0,C 180,E1 -3318.484,E2 -3318.484} C_VEL
LIN {X 0,Y 552.486,Z 426.82,A -85,B 0,C 180,E1 -3319.093,E2 -3319.093} C_VEL
LIN {X 0,Y 552.327,Z 436.435,A -85,B 0,C 180,E1 -3319.831,E2 -3319.831} C_VEL
LIN {X 0,Y 552.153,Z 447.105,A -85,B 0,C 180,E1 -3320.845,E2 -3320.845} C_VEL
LIN {X 0,Y 552.01,Z 454.905,A -85,B 0,C 180,E1 -3321.765,E2 -3321.765} C_VEL
LIN {X 0,Y 551.904,Z 461.415,A -85,B 0,C 180,E1 -3322.684,E2 -3322.684} C_VEL
LIN {X 0,Y 551.809,Z 467.105,A -85,B 0,C 180,E1 -3323.651,E2 -3323.651} C_VEL
LIN {X 0,Y 551.802,Z 471.352,A -85,B 0,C 180,E1 -3324.519,E2 -3324.519} C_VEL
LIN {X 0,Y 551.767,Z 475.643,A -85,B 0,C 180,E1 -3325.617,E2 -3325.617} C_VEL
LIN {X 0,Y 551.75,Z 477.975,A -85,B 0,C 180,E1 -3326.348,E2 -3326.348} C_VEL
LIN {X 0,Y 551.723,Z 479.773,A -85,B 0,C 180,E1 -3327.079,E2 -3327.079} C_VEL
LIN {X 0,Y 551.645,Z 482.196,A -85,B 0,C 180,E1 -3328.54,E2 -3328.54} C_VEL
LIN {X 0,Y 551.641,Z 482.78,A -85,B 0,C 180,E1 -3329.27,E2 -3329.27} C_VEL
LIN {X 0,Y 551.641,Z 482.78,A -85,B 0,C 180,E1 -3330.73,E2 -3330.73} C_VEL
LIN {X 0,Y 551.645,Z 482.196,A -85,B 0,C 180,E1 -3331.46,E2 -3331.46} C_VEL
LIN {X 0,Y 551.723,Z 479.773,A -85,B 0,C 180,E1 -3332.921,E2 -3332.921} C_VEL
LIN {X 0,Y 551.764,Z 476.852,A -85,B 0,C 180,E1 -3334.017,E2 -3334.017} C_VEL
LIN {X 0,Y 551.723,Z 472.896,A -85,B 0,C 180,E1 -3335.116,E2 -3335.116} C_VEL
LIN {X 0,Y 551.837,Z 468.403,A -85,B 0,C 180,E1 -3336.098,E2 -3336.098} C_VEL
LIN {X 0,Y 551.886,Z 462.565,A -85,B 0,C 180,E1 -3337.132,E2 -3337.132} C_VEL
LIN {X 0,Y 551.984,Z 456.275,A -85,B 0,C 180,E1 -3338.051,E2 -3338.051} C_VEL
LIN {X 0,Y 552.122,Z 448.728,A -85,B 0,C 180,E1 -3338.971,E2 -3338.971} C_VEL
LIN {X 0,Y 552.28,Z 439.619,A -85,B 0,C 180,E1 -3339.892,E2 -3339.892} C_VEL
LIN {X 0,Y 552.47,Z 428.169,A -85,B 0,C 180,E1 -3340.815,E2 -3340.815} C_VEL
LIN {X 0,Y 552.569,Z 419.426,A -85,B 0,C 180,E1 -3341.389,E2 -3341.389} C_VEL
LIN {X 0,Y 552.743,Z 408.387,A -85,B 0,C 180,E1 -3341.971,E2 -3341.971} C_VEL
LIN {X 0,Y 552.885,Z 398.321,A -85,B 0,C 180,E1 -3342.387,E2 -3342.387} C_VEL
LIN {X 0,Y 553.03,Z 387.964,A -85,B 0,C 180,E1 -3342.71,E2 -3342.71} C_VEL
LIN {X 0,Y 552.737,Z 383.526,A -85,B 0,C 180,E1 -3342.833,E2 -3342.833} C_VEL
LIN {X 0,Y 551.73,Z 377.523,A -85,B 0,C 180,E1 -3342.974,E2 -3342.974} C_VEL
LIN {X 0,Y 551.766,Z 371.46,A -85,B 0,C 180,E1 -3345.514,E2 -3345.514} C_VEL
LIN {X 0,Y 551.821,Z 366.061,A -85,B 0,C 180,E1 -3347.798,E2 -3347.798} C_VEL
LIN {X 0,Y 551.86,Z 360.582,A -85,B 0,C 180,E1 -3350.111,E2 -3350.111} C_VEL
LIN {X 0,Y 551.88,Z 355.104,A -85,B 0,C 180,E1 -3352.46,E2 -3352.46} C_VEL
LIN {X 0,Y 551.994,Z 348.09,A -85,B 0,C 180,E1 -3355.651,E2 -3355.651} C_VEL
LIN {X 0,Y 552.084,Z 341.885,A -85,B 0,C 180,E1 -3358.554,E2 -3358.554} C_VEL
LIN {X 0,Y 552.146,Z 337.684,A -85,B 0,C 180,E1 -3360.606,E2 -3360.606} C_VEL
LIN {X 0,Y 552.245,Z 332.646,A -85,B 0,C 180,E1 -3363.177,E2 -3363.177} C_VEL
LIN {X 0,Y 552.355,Z 327.703,A -85,B 0,C 180,E1 -3365.823,E2 -3365.823} C_VEL
LIN {X 0,Y 552.466,Z 322.9,A -85,B 0,C 180,E1 -3368.56,E2 -3368.56} C_VEL
LIN {X 0,Y 552.528,Z 318.238,A -85,B 0,C 180,E1 -3371.408,E2 -3371.408} C_VEL
LIN {X 0,Y 552.386,Z 315.046,A -85,B 0,C 180,E1 -3373.513,E2 -3373.513} C_VEL
LIN {X 0,Y 552.151,Z 313.602,A -85,B 0,C 180,E1 -3374.537,E2 -3374.537} C_VEL
LIN {X 0,Y 552.097,Z 313.215,A -85,B 0,C 180,E1 -3375.562,E2 -3375.562} C_VEL
LIN {X 0,Y 552.122,Z 313.212,A -85,B 0,C 180,E1 -3378.554,E2 -3378.554} C_VEL
LIN {X 0,Y 552.12,Z 313.208,A -85,B 0,C 180,E1 -3381.411,E2 -3381.411} C_VEL
LIN {X 0,Y 552.086,Z 313.219,A -85,B 0,C 180,E1 -3384.156,E2 -3384.156} C_VEL
LIN {X 0,Y 552.116,Z 313.206,A -85,B 0,C 180,E1 -3386.814,E2 -3386.814} C_VEL
LIN {X 0,Y 552.102,Z 313.21,A -85,B 0,C 180,E1 -3389.39,E2 -3389.39} C_VEL
LIN {X 0,Y 552.11,Z 313.215,A -85,B 0,C 180,E1 -3391.901,E2 -3391.901} C_VEL
LIN {X 0,Y 552.156,Z 313.201,A -85,B 0,C 180,E1 -3394.649,E2 -3394.649} C_VEL
LIN {X 0,Y 552.092,Z 313.215,A -85,B 0,C 180,E1 -3397.549,E2 -3397.549} C_VEL
LIN {X 0,Y 552.144,Z 313.203,A -85,B 0,C 180,E1 -3400.375,E2 -3400.375} C_VEL
LIN {X 0,Y 552.155,Z 313.202,A -85,B 0,C 180,E1 -3402.977,E2 -3402.977} C_VEL
LIN {X 0,Y 552.135,Z 313.206,A -85,B 0,C 180,E1 -3406.004,E2 -3406.004} C_VEL
LIN {X 0,Y 552.163,Z 313.203,A -85,B 0,C 180,E1 -3408.993,E2 -3408.993} C_VEL
LIN {X 0,Y 552.157,Z 313.202,A -85,B 0,C 180,E1 -3411.951,E2 -3411.951} C_VEL
LIN {X 0,Y 552.229,Z 313.195,A -85,B 0,C 180,E1 -3414.889,E2 -3414.889} C_VEL
LIN {X 0,Y 552.227,Z 313.193,A -85,B 0,C 180,E1 -3417.812,E2 -3417.812} C_VEL
LIN {X 0,Y 552.239,Z 313.194,A -85,B 0,C 180,E1 -3420.729,E2 -3420.729} C_VEL
LIN {X 0,Y 552.202,Z 313.201,A -85,B 0,C 180,E1 -3422.918,E2 -3422.918} C_VEL
LIN {X 0,Y 552.202,Z 313.195,A -85,B 0,C 180,E1 -3425.843,E2 -3425.843} C_VEL
LIN {X 0,Y 552.156,Z 313.207,A -85,B 0,C 180,E1 -3428.785,E2 -3428.785} C_VEL
LIN {X 0,Y 552.161,Z 313.2,A -85,B 0,C 180,E1 -3431.75,E2 -3431.75} C_VEL
LIN {X 0,Y 552.135,Z 313.212,A -85,B 0,C 180,E1 -3434.748,E2 -3434.748} C_VEL
LIN {X 0,Y 552.108,Z 313.207,A -85,B 0,C 180,E1 -3437.788,E2 -3437.788} C_VEL
LIN {X 0,Y 552.129,Z 313.206,A -85,B 0,C 180,E1 -3440.101,E2 -3440.101} C_VEL
LIN {X 0,Y 552.091,Z 313.215,A -85,B 0,C 180,E1 -3442.451,E2 -3442.451} C_VEL
LIN {X 0,Y 552.153,Z 313.201,A -85,B 0,C 180,E1 -3445.35,E2 -3445.35} C_VEL
LIN {X 0,Y 552.117,Z 313.209,A -85,B 0,C 180,E1 -3448.097,E2 -3448.097} C_VEL
LIN {X 0,Y 552.105,Z 313.214,A -85,B 0,C 180,E1 -3450.609,E2 -3450.609} C_VEL
LIN {X 0,Y 552.12,Z 313.205,A -85,B 0,C 180,E1 -3453.185,E2 -3453.185} C_VEL
LIN {X 0,Y 552.11,Z 313.208,A -85,B 0,C 180,E1 -3453.782,E2 -3453.782} C_VEL
LIN {X 0,Y 551.472,Z 313.295,A -85,B 0,C 180,E1 -3454.39,E2 -3454.39} C_VEL
LIN {X 0,Y 548.651,Z 313.645,A -85,B 0,C 180,E1 -3455.379,E2 -3455.379} C_VEL
LIN {X 0,Y 546.233,Z 313.946,A -85,B 0,C 180,E1 -3456.174,E2 -3456.174} C_VEL
LIN {X 0,Y 545.164,Z 314.074,A -85,B 0,C 180,E1 -3456.788,E2 -3456.788} C_VEL
LIN {X 0,Y 545.062,Z 314.085,A -85,B 0,C 180,E1 -3456.996,E2 -3456.996} C_VEL
LIN {X 0,Y 545.09,Z 314.089,A -85,B 0,C 180,E1 -3460.14,E2 -3460.14} C_VEL
LIN {X 0,Y 545.083,Z 314.082,A -85,B 0,C 180,E1 -3463.105,E2 -3463.105} C_VEL
LIN {X 0,Y 545.056,Z 314.092,A -85,B 0,C 180,E1 -3466.225,E2 -3466.225} C_VEL
LIN {X 0,Y 545.098,Z 314.08,A -85,B 0,C 180,E1 -3468.887,E2 -3468.887} C_VEL
LIN {X 0,Y 545.052,Z 314.093,A -85,B 0,C 180,E1 -3471.763,E2 -3471.763} C_VEL
LIN {X 0,Y 545.049,Z 314.087,A -85,B 0,C 180,E1 -3474.533,E2 -3474.533} C_VEL
LIN {X 0,Y 545.078,Z 314.084,A -85,B 0,C 180,E1 -3477.212,E2 -3477.212} C_VEL
LIN {X 0,Y 545.063,Z 314.093,A -85,B 0,C 180,E1 -3479.811,E2 -3479.811} C_VEL
LIN {X 0,Y 545.093,Z 314.082,A -85,B 0,C 180,E1 -3482.345,E2 -3482.345} C_VEL
LIN {X 0,Y 545.115,Z 314.078,A -85,B 0,C 180,E1 -3484.82,E2 -3484.82} C_VEL
LIN {X 0,Y 545.035,Z 314.092,A -85,B 0,C 180,E1 -3487.242,E2 -3487.242} C_VEL
LIN {X 0,Y 545.117,Z 314.078,A -85,B 0,C 180,E1 -3490.415,E2 -3490.415} C_VEL
LIN {X 0,Y 545.071,Z 314.092,A -85,B 0,C 180,E1 -3493.521,E2 -3493.521} C_VEL
LIN {X 0,Y 545.092,Z 314.085,A -85,B 0,C 180,E1 -3495.82,E2 -3495.82} C_VEL
LIN {X 0,Y 545.116,Z 314.082,A -85,B 0,C 180,E1 -3498.849,E2 -3498.849} C_VEL
LIN {X 0,Y 545.127,Z 314.079,A -85,B 0,C 180,E1 -3501.847,E2 -3501.847} C_VEL
LIN {X 0,Y 545.204,Z 314.073,A -85,B 0,C 180,E1 -3504.823,E2 -3504.823} C_VEL
LIN {X 0,Y 545.197,Z 314.07,A -85,B 0,C 180,E1 -3507.784,E2 -3507.784} C_VEL
LIN {X 0,Y 545.21,Z 314.073,A -85,B 0,C 180,E1 -3510.739,E2 -3510.739} C_VEL
LIN {X 0,Y 545.169,Z 314.08,A -85,B 0,C 180,E1 -3512.956,E2 -3512.956} C_VEL
LIN {X 0,Y 545.177,Z 314.072,A -85,B 0,C 180,E1 -3515.919,E2 -3515.919} C_VEL
LIN {X 0,Y 545.118,Z 314.086,A -85,B 0,C 180,E1 -3518.9,E2 -3518.9} C_VEL
LIN {X 0,Y 545.132,Z 314.077,A -85,B 0,C 180,E1 -3521.904,E2 -3521.904} C_VEL
LIN {X 0,Y 545.082,Z 314.088,A -85,B 0,C 180,E1 -3524.944,E2 -3524.944} C_VEL
LIN {X 0,Y 545.077,Z 314.086,A -85,B 0,C 180,E1 -3528.026,E2 -3528.026} C_VEL
LIN {X 0,Y 545.093,Z 314.088,A -85,B 0,C 180,E1 -3530.372,E2 -3530.372} C_VEL
LIN {X 0,Y 545.078,Z 314.082,A -85,B 0,C 180,E1 -3533.559,E2 -3533.559} C_VEL
LIN {X 0,Y 545.086,Z 314.085,A -85,B 0,C 180,E1 -3536,E2 -3536} C_VEL
LIN {X 0,Y 545.087,Z 314.084,A -85,B 0,C 180,E1 -3538.749,E2 -3538.749} C_VEL
LIN {X 0,Y 545.075,Z 314.085,A -85,B 0,C 180,E1 -3541.683,E2 -3541.683} C_VEL
LIN {X 0,Y 545.073,Z 314.086,A -85,B 0,C 180,E1 -3544.563,E2 -3544.563} C_VEL
LIN {X 0,Y 545.036,Z 314.088,A -85,B 0,C 180,E1 -3547.304,E2 -3547.304} C_VEL
LIN {X 0,Y 545.09,Z 314.089,A -85,B 0,C 180,E1 -3550.14,E2 -3550.14} C_VEL
LIN {X 0,Y 545.078,Z 314.083,A -85,B 0,C 180,E1 -3553.106,E2 -3553.106} C_VEL
LIN {X 0,Y 545.061,Z 314.089,A -85,B 0,C 180,E1 -3556.225,E2 -3556.225} C_VEL
LIN {X 0,Y 545.098,Z 314.08,A -85,B 0,C 180,E1 -3558.888,E2 -3558.888} C_VEL
LIN {X 0,Y 545.052,Z 314.095,A -85,B 0,C 180,E1 -3561.763,E2 -3561.763} C_VEL
LIN {X 0,Y 545.033,Z 314.088,A -85,B 0,C 180,E1 -3564.532,E2 -3564.532} C_VEL
LIN {X 0,Y 545.079,Z 314.086,A -85,B 0,C 180,E1 -3567.213,E2 -3567.213} C_VEL
LIN {X 0,Y 545.063,Z 314.09,A -85,B 0,C 180,E1 -3569.811,E2 -3569.811} C_VEL
LIN {X 0,Y 545.086,Z 314.082,A -85,B 0,C 180,E1 -3572.345,E2 -3572.345} C_VEL
LIN {X 0,Y 545.115,Z 314.079,A -85,B 0,C 180,E1 -3574.821,E2 -3574.821} C_VEL
LIN {X 0,Y 545.037,Z 314.095,A -85,B 0,C 180,E1 -3577.243,E2 -3577.243} C_VEL
LIN {X 0,Y 545.118,Z 314.077,A -85,B 0,C 180,E1 -3580.415,E2 -3580.415} C_VEL
LIN {X 0,Y 545.07,Z 314.088,A -85,B 0,C 180,E1 -3583.522,E2 -3583.522} C_VEL
LIN {X 0,Y 545.093,Z 314.082,A -85,B 0,C 180,E1 -3585.82,E2 -3585.82} C_VEL
LIN {X 0,Y 545.116,Z 314.083,A -85,B 0,C 180,E1 -3588.85,E2 -3588.85} C_VEL
LIN {X 0,Y 545.127,Z 314.077,A -85,B 0,C 180,E1 -3591.847,E2 -3591.847} C_VEL
LIN {X 0,Y 545.203,Z 314.074,A -85,B 0,C 180,E1 -3594.823,E2 -3594.823} C_VEL
LIN {X 0,Y 545.197,Z 314.068,A -85,B 0,C 180,E1 -3597.784,E2 -3597.784} C_VEL
LIN {X 0,Y 545.214,Z 314.074,A -85,B 0,C 180,E1 -3600.739,E2 -3600.739} C_VEL
LIN {X 0,Y 545.17,Z 314.077,A -85,B 0,C 180,E1 -3602.956,E2 -3602.956} C_VEL
LIN {X 0,Y 545.171,Z 314.071,A -85,B 0,C 180,E1 -3605.92,E2 -3605.92} C_VEL
LIN {X 0,Y 545.12,Z 314.082,A -85,B 0,C 180,E1 -3608.9,E2 -3608.9} C_VEL
LIN {X 0,Y 545.134,Z 314.077,A -85,B 0,C 180,E1 -3611.905,E2 -3611.905} C_VEL
LIN {X 0,Y 545.086,Z 314.084,A -85,B 0,C 180,E1 -3614.944,E2 -3614.944} C_VEL
LIN {X 0,Y 545.071,Z 314.087,A -85,B 0,C 180,E1 -3618.026,E2 -3618.026} C_VEL
LIN {X 0,Y 545.092,Z 314.09,A -85,B 0,C 180,E1 -3620.373,E2 -3620.373} C_VEL
LIN {X 0,Y 545.079,Z 314.083,A -85,B 0,C 180,E1 -3623.56,E2 -3623.56} C_VEL
LIN {X 0,Y 545.08,Z 314.089,A -85,B 0,C 180,E1 -3626.001,E2 -3626.001} C_VEL
LIN {X 0,Y 545.089,Z 314.082,A -85,B 0,C 180,E1 -3628.748,E2 -3628.748} C_VEL
LIN {X 0,Y 545.058,Z 314.089,A -85,B 0,C 180,E1 -3631.679,E2 -3631.679} C_VEL
LIN {X 0,Y 545.062,Z 314.086,A -85,B 0,C 180,E1 -3634.565,E2 -3634.565} C_VEL
LIN {X 0,Y 545.037,Z 314.091,A -85,B 0,C 180,E1 -3637.304,E2 -3637.304} C_VEL
LIN {X 0,Y 545.069,Z 314.091,A -85,B 0,C 180,E1 -3640.143,E2 -3640.143} C_VEL
LIN {X 0,Y 545.079,Z 314.087,A -85,B 0,C 180,E1 -3643.107,E2 -3643.107} C_VEL
LIN {X 0,Y 545.052,Z 314.093,A -85,B 0,C 180,E1 -3644.832,E2 -3644.832} C_VEL
LIN {X 0,Y 545.509,Z 317.393,A -85,B 0,C 180,E1 -3647.253,E2 -3647.253} C_VEL
LIN {X 0,Y 545.525,Z 321.509,A -85,B 0,C 180,E1 -3649.898,E2 -3649.898} C_VEL
LIN {X 0,Y 545.44,Z 326.222,A -85,B 0,C 180,E1 -3652.729,E2 -3652.729} C_VEL
LIN {X 0,Y 545.28,Z 331.318,A -85,B 0,C 180,E1 -3655.577,E2 -3655.577} C_VEL
LIN {X 0,Y 545.176,Z 336.474,A -85,B 0,C 180,E1 -3658.302,E2 -3658.302} C_VEL
LIN {X 0,Y 545.055,Z 342.389,A -85,B 0,C 180,E1 -3661.259,E2 -3661.259} C_VEL
LIN {X 0,Y 544.944,Z 348.091,A -85,B 0,C 180,E1 -3663.993,E2 -3663.993} C_VEL
LIN {X 0,Y 544.838,Z 353.348,A -85,B 0,C 180,E1 -3666.43,E2 -3666.43} C_VEL
LIN {X 0,Y 544.795,Z 358.66,A -85,B 0,C 180,E1 -3668.826,E2 -3668.826} C_VEL
LIN {X 0,Y 544.748,Z 364.144,A -85,B 0,C 180,E1 -3671.184,E2 -3671.184} C_VEL
LIN {X 0,Y 544.69,Z 369.615,A -85,B 0,C 180,E1 -3673.509,E2 -3673.509} C_VEL
LIN {X 0,Y 544.687,Z 375.053,A -85,B 0,C 180,E1 -3675.809,E2 -3675.809} C_VEL
LIN {X 0,Y 544.631,Z 377.523,A -85,B 0,C 180,E1 -3676.854,E2 -3676.854} C_VEL
LIN {X 0,Y 546.091,Z 387.06,A -85,B 0,C 180,E1 -3677.103,E2 -3677.103} C_VEL
LIN {X 0,Y 545.988,Z 397.017,A -85,B 0,C 180,E1 -3677.407,E2 -3677.407} C_VEL
LIN {X 0,Y 545.828,Z 407.364,A -85,B 0,C 180,E1 -3677.828,E2 -3677.828} C_VEL
LIN {X 0,Y 545.628,Z 417.155,A -85,B 0,C 180,E1 -3678.334,E2 -3678.334} C_VEL
LIN {X 0,Y 545.496,Z 425.457,A -85,B 0,C 180,E1 -3678.857,E2 -3678.857} C_VEL
LIN {X 0,Y 545.379,Z 434.16,A -85,B 0,C 180,E1 -3679.513,E2 -3679.513} C_VEL
LIN {X 0,Y 545.225,Z 441.53,A -85,B 0,C 180,E1 -3680.166,E2 -3680.166} C_VEL
LIN {X 0,Y 545.1,Z 448.721,A -85,B 0,C 180,E1 -3680.913,E2 -3680.913} C_VEL
LIN {X 0,Y 544.92,Z 456.267,A -85,B 0,C 180,E1 -3681.844,E2 -3681.844} C_VEL
LIN {X 0,Y 544.822,Z 462.556,A -85,B 0,C 180,E1 -3682.775,E2 -3682.775} C_VEL
LIN {X 0,Y 544.758,Z 468.648,A -85,B 0,C 180,E1 -3683.872,E2 -3683.872} C_VEL
LIN {X 0,Y 544.64,Z 474.388,A -85,B 0,C 180,E1 -3685.189,E2 -3685.189} C_VEL
LIN {X 0,Y 544.669,Z 477.975,A -85,B 0,C 180,E1 -3686.301,E2 -3686.301} C_VEL
LIN {X 0,Y 544.65,Z 479.768,A -85,B 0,C 180,E1 -3687.041,E2 -3687.041} C_VEL
LIN {X 0,Y 544.546,Z 482.195,A -85,B 0,C 180,E1 -3688.521,E2 -3688.521} C_VEL
LIN {X 0,Y 544.542,Z 482.779,A -85,B 0,C 180,E1 -3689.261,E2 -3689.261} C_VEL
LIN {X 0,Y 544.542,Z 482.779,A -85,B 0,C 180,E1 -3690.739,E2 -3690.739} C_VEL
LIN {X 0,Y 544.546,Z 482.195,A -85,B 0,C 180,E1 -3691.479,E2 -3691.479} C_VEL
LIN {X 0,Y 544.65,Z 479.768,A -85,B 0,C 180,E1 -3692.959,E2 -3692.959} C_VEL
LIN {X 0,Y 544.684,Z 476.845,A -85,B 0,C 180,E1 -3694.069,E2 -3694.069} C_VEL
LIN {X 0,Y 544.653,Z 472.888,A -85,B 0,C 180,E1 -3695.182,E2 -3695.182} C_VEL
LIN {X 0,Y 544.759,Z 468.646,A -85,B 0,C 180,E1 -3696.129,E2 -3696.129} C_VEL
LIN {X 0,Y 544.822,Z 462.556,A -85,B 0,C 180,E1 -3697.225,E2 -3697.225} C_VEL
LIN {X 0,Y 544.92,Z 456.267,A -85,B 0,C 180,E1 -3698.156,E2 -3698.156} C_VEL
LIN {X 0,Y 545.1,Z 448.721,A -85,B 0,C 180,E1 -3699.087,E2 -3699.087} C_VEL
LIN {X 0,Y 545.276,Z 439.614,A -85,B 0,C 180,E1 -3700.02,E2 -3700.02} C_VEL
LIN {X 0,Y 545.465,Z 428.155,A -85,B 0,C 180,E1 -3700.955,E2 -3700.955} C_VEL
LIN {X 0,Y 545.603,Z 418.394,A -85,B 0,C 180,E1 -3701.595,E2 -3701.595} C_VEL
LIN {X 0,Y 545.793,Z 408.37,A -85,B 0,C 180,E1 -3702.125,E2 -3702.125} C_VEL
LIN {X 0,Y 545.938,Z 398.303,A -85,B 0,C 180,E1 -3702.547,E2 -3702.547} C_VEL
LIN {X 0,Y 546.092,Z 387.934,A -85,B 0,C 180,E1 -3702.874,E2 -3702.874} C_VEL
LIN {X 0,Y 545.614,Z 383.272,A -85,B 0,C 180,E1 -3703.009,E2 -3703.009} C_VEL
LIN {X 0,Y 544.631,Z 377.523,A -85,B 0,C 180,E1 -3703.146,E2 -3703.146} C_VEL
LIN {X 0,Y 544.672,Z 371.436,A -85,B 0,C 180,E1 -3705.722,E2 -3705.722} C_VEL
LIN {X 0,Y 544.731,Z 365.969,A -85,B 0,C 180,E1 -3708.038,E2 -3708.038} C_VEL
LIN {X 0,Y 544.796,Z 360.49,A -85,B 0,C 180,E1 -3710.384,E2 -3710.384} C_VEL
LIN {X 0,Y 544.824,Z 355.102,A -85,B 0,C 180,E1 -3712.767,E2 -3712.767} C_VEL
LIN {X 0,Y 544.933,Z 349.229,A -85,B 0,C 180,E1 -3715.472,E2 -3715.472} C_VEL
LIN {X 0,Y 545.027,Z 342.846,A -85,B 0,C 180,E1 -3718.496,E2 -3718.496} C_VEL
LIN {X 0,Y 545.123,Z 337.744,A -85,B 0,C 180,E1 -3721.044,E2 -3721.044} C_VEL
LIN {X 0,Y 545.231,Z 332.713,A -85,B 0,C 180,E1 -3723.66,E2 -3723.66} C_VEL
LIN {X 0,Y 545.351,Z 327.82,A -85,B 0,C 180,E1 -3726.356,E2 -3726.356} C_VEL
LIN {X 0,Y 545.497,Z 322.675,A -85,B 0,C 180,E1 -3729.374,E2 -3729.374} C_VEL
LIN {X 0,Y 545.536,Z 318.422,A -85,B 0,C 180,E1 -3732.059,E2 -3732.059} C_VEL
LIN {X 0,Y 545.252,Z 315.438,A -85,B 0,C 180,E1 -3734.109,E2 -3734.109} C_VEL
LIN {X 0,Y 545.052,Z 314.092,A -85,B 0,C 180,E1 -3735.168,E2 -3735.168} C_VEL
LIN {X 0,Y 545.078,Z 314.09,A -85,B 0,C 180,E1 -3737.897,E2 -3737.897} C_VEL
LIN {X 0,Y 545.084,Z 314.085,A -85,B 0,C 180,E1 -3740.818,E2 -3740.818} C_VEL
LIN {X 0,Y 545.042,Z 314.092,A -85,B 0,C 180,E1 -3743.619,E2 -3743.619} C_VEL
LIN {X 0,Y 545.066,Z 314.088,A -85,B 0,C 180,E1 -3746.328,E2 -3746.328} C_VEL
LIN {X 0,Y 545.066,Z 314.084,A -85,B 0,C 180,E1 -3748.952,E2 -3748.952} C_VEL
LIN {X 0,Y 545.102,Z 314.083,A -85,B 0,C 180,E1 -3751.507,E2 -3751.507} C_VEL
LIN {X 0,Y 545.095,Z 314.081,A -85,B 0,C 180,E1 -3754.491,E2 -3754.491} C_VEL
LIN {X 0,Y 545.037,Z 314.09,A -85,B 0,C 180,E1 -3757.242,E2 -3757.242} C_VEL
LIN {X 0,Y 545.116,Z 314.078,A -85,B 0,C 180,E1 -3760.414,E2 -3760.414} C_VEL
LIN {X 0,Y 545.073,Z 314.092,A -85,B 0,C 180,E1 -3763.521,E2 -3763.521} C_VEL
LIN {X 0,Y 545.094,Z 314.085,A -85,B 0,C 180,E1 -3765.82,E2 -3765.82} C_VEL
LIN {X 0,Y 545.118,Z 314.079,A -85,B 0,C 180,E1 -3768.849,E2 -3768.849} C_VEL
LIN {X 0,Y 545.128,Z 314.079,A -85,B 0,C 180,E1 -3771.847,E2 -3771.847} C_VEL
LIN {X 0,Y 545.205,Z 314.069,A -85,B 0,C 180,E1 -3774.823,E2 -3774.823} C_VEL
LIN {X 0,Y 545.198,Z 314.069,A -85,B 0,C 180,E1 -3777.783,E2 -3777.783} C_VEL
LIN {X 0,Y 545.209,Z 314.069,A -85,B 0,C 180,E1 -3780.738,E2 -3780.738} C_VEL
LIN {X 0,Y 545.17,Z 314.078,A -85,B 0,C 180,E1 -3782.955,E2 -3782.955} C_VEL
LIN {X 0,Y 545.172,Z 314.071,A -85,B 0,C 180,E1 -3785.919,E2 -3785.919} C_VEL
LIN {X 0,Y 545.115,Z 314.086,A -85,B 0,C 180,E1 -3788.9,E2 -3788.9} C_VEL
LIN {X 0,Y 545.133,Z 314.075,A -85,B 0,C 180,E1 -3791.904,E2 -3791.904} C_VEL
LIN {X 0,Y 545.084,Z 314.089,A -85,B 0,C 180,E1 -3794.943,E2 -3794.943} C_VEL
LIN {X 0,Y 545.077,Z 314.083,A -85,B 0,C 180,E1 -3798.025,E2 -3798.025} C_VEL
LIN {X 0,Y 545.093,Z 314.085,A -85,B 0,C 180,E1 -3800.372,E2 -3800.372} C_VEL
LIN {X 0,Y 545.079,Z 314.082,A -85,B 0,C 180,E1 -3803.559,E2 -3803.559} C_VEL
LIN {X 0,Y 545.078,Z 314.084,A -85,B 0,C 180,E1 -3806,E2 -3806} C_VEL
LIN {X 0,Y 545.087,Z 314.087,A -85,B 0,C 180,E1 -3808.748,E2 -3808.748} C_VEL
LIN {X 0,Y 545.076,Z 314.083,A -85,B 0,C 180,E1 -3811.682,E2 -3811.682} C_VEL
LIN {X 0,Y 545.073,Z 314.089,A -85,B 0,C 180,E1 -3814.563,E2 -3814.563} C_VEL
LIN {X 0,Y 545.062,Z 314.085,A -85,B 0,C 180,E1 -3816.996,E2 -3816.996} C_VEL
LIN {X 0,Y 544.357,Z 314.174,A -85,B 0,C 180,E1 -3817.612,E2 -3817.612} C_VEL
LIN {X 0,Y 541.503,Z 314.532,A -85,B 0,C 180,E1 -3818.613,E2 -3818.613} C_VEL
LIN {X 0,Y 539.126,Z 314.827,A -85,B 0,C 180,E1 -3819.419,E2 -3819.419} C_VEL
LIN {X 0,Y 538.12,Z 314.956,A -85,B 0,C 180,E1 -3820.041,E2 -3820.041} C_VEL
LIN {X 0,Y 538.044,Z 314.959,A -85,B 0,C 180,E1 -3820.252,E2 -3820.252} C_VEL
LIN {X 0,Y 538.03,Z 314.961,A -85,B 0,C 180,E1 -3822.988,E2 -3822.988} C_VEL
LIN {X 0,Y 538.023,Z 314.968,A -85,B 0,C 180,E1 -3825.926,E2 -3825.926} C_VEL
LIN {X 0,Y 538.075,Z 314.955,A -85,B 0,C 180,E1 -3829.249,E2 -3829.249} C_VEL
LIN {X 0,Y 537.991,Z 314.971,A -85,B 0,C 180,E1 -3832.122,E2 -3832.122} C_VEL
LIN {X 0,Y 538.009,Z 314.963,A -85,B 0,C 180,E1 -3834.917,E2 -3834.917} C_VEL
LIN {X 0,Y 538.028,Z 314.967,A -85,B 0,C 180,E1 -3837.618,E2 -3837.618} C_VEL
LIN {X 0,Y 538.015,Z 314.964,A -85,B 0,C 180,E1 -3840.239,E2 -3840.239} C_VEL
LIN {X 0,Y 538.068,Z 314.956,A -85,B 0,C 180,E1 -3842.797,E2 -3842.797} C_VEL
LIN {X 0,Y 538.046,Z 314.963,A -85,B 0,C 180,E1 -3845.293,E2 -3845.293} C_VEL
LIN {X 0,Y 538.019,Z 314.962,A -85,B 0,C 180,E1 -3848.546,E2 -3848.546} C_VEL
LIN {X 0,Y 538.035,Z 314.962,A -85,B 0,C 180,E1 -3850.94,E2 -3850.94} C_VEL
LIN {X 0,Y 538.022,Z 314.97,A -85,B 0,C 180,E1 -3853.299,E2 -3853.299} C_VEL
LIN {X 0,Y 538.061,Z 314.963,A -85,B 0,C 180,E1 -3855.631,E2 -3855.631} C_VEL
LIN {X 0,Y 538.075,Z 314.958,A -85,B 0,C 180,E1 -3858.702,E2 -3858.702} C_VEL
LIN {X 0,Y 538.084,Z 314.957,A -85,B 0,C 180,E1 -3861.74,E2 -3861.74} C_VEL
LIN {X 0,Y 538.162,Z 314.949,A -85,B 0,C 180,E1 -3864.755,E2 -3864.755} C_VEL
LIN {X 0,Y 538.168,Z 314.945,A -85,B 0,C 180,E1 -3867.755,E2 -3867.755} C_VEL
LIN {X 0,Y 538.18,Z 314.949,A -85,B 0,C 180,E1 -3870.748,E2 -3870.748} C_VEL
LIN {X 0,Y 538.136,Z 314.956,A -85,B 0,C 180,E1 -3872.994,E2 -3872.994} C_VEL
LIN {X 0,Y 538.131,Z 314.95,A -85,B 0,C 180,E1 -3875.997,E2 -3875.997} C_VEL
LIN {X 0,Y 538.069,Z 314.963,A -85,B 0,C 180,E1 -3879.018,E2 -3879.018} C_VEL
LIN {X 0,Y 538.08,Z 314.956,A -85,B 0,C 180,E1 -3882.063,E2 -3882.063} C_VEL
LIN {X 0,Y 538.042,Z 314.963,A -85,B 0,C 180,E1 -3885.144,E2 -3885.144} C_VEL
LIN {X 0,Y 538.029,Z 314.967,A -85,B 0,C 180,E1 -3888.27,E2 -3888.27} C_VEL
LIN {X 0,Y 538.036,Z 314.967,A -85,B 0,C 180,E1 -3890.651,E2 -3890.651} C_VEL
LIN {X 0,Y 538.001,Z 314.966,A -85,B 0,C 180,E1 -3893.888,E2 -3893.888} C_VEL
LIN {X 0,Y 538.047,Z 314.968,A -85,B 0,C 180,E1 -3896.366,E2 -3896.366} C_VEL
LIN {X 0,Y 538.028,Z 314.962,A -85,B 0,C 180,E1 -3898.934,E2 -3898.934} C_VEL
LIN {X 0,Y 538.025,Z 314.965,A -85,B 0,C 180,E1 -3901.89,E2 -3901.89} C_VEL
LIN {X 0,Y 538.023,Z 314.964,A -85,B 0,C 180,E1 -3904.62,E2 -3904.62} C_VEL
LIN {X 0,Y 538.004,Z 314.964,A -85,B 0,C 180,E1 -3907.171,E2 -3907.171} C_VEL
LIN {X 0,Y 538.051,Z 314.963,A -85,B 0,C 180,E1 -3909.794,E2 -3909.794} C_VEL
LIN {X 0,Y 538.017,Z 314.962,A -85,B 0,C 180,E1 -3912.786,E2 -3912.786} C_VEL
LIN {X 0,Y 538.026,Z 314.97,A -85,B 0,C 180,E1 -3915.926,E2 -3915.926} C_VEL
LIN {X 0,Y 538.075,Z 314.957,A -85,B 0,C 180,E1 -3919.249,E2 -3919.249} C_VEL
LIN {X 0,Y 537.991,Z 314.969,A -85,B 0,C 180,E1 -3922.123,E2 -3922.123} C_VEL
LIN {X 0,Y 537.995,Z 314.965,A -85,B 0,C 180,E1 -3924.916,E2 -3924.916} C_VEL
LIN {X 0,Y 538.029,Z 314.97,A -85,B 0,C 180,E1 -3927.619,E2 -3927.619} C_VEL
LIN {X 0,Y 538.016,Z 314.963,A -85,B 0,C 180,E1 -3930.239,E2 -3930.239} C_VEL
LIN {X 0,Y 538.061,Z 314.958,A -85,B 0,C 180,E1 -3932.797,E2 -3932.797} C_VEL
LIN {X 0,Y 538.046,Z 314.966,A -85,B 0,C 180,E1 -3935.293,E2 -3935.293} C_VEL
LIN {X 0,Y 538.02,Z 314.962,A -85,B 0,C 180,E1 -3938.546,E2 -3938.546} C_VEL
LIN {X 0,Y 538.035,Z 314.964,A -85,B 0,C 180,E1 -3940.94,E2 -3940.94} C_VEL
LIN {X 0,Y 538.022,Z 314.97,A -85,B 0,C 180,E1 -3943.299,E2 -3943.299} C_VEL
LIN {X 0,Y 538.062,Z 314.959,A -85,B 0,C 180,E1 -3945.631,E2 -3945.631} C_VEL
LIN {X 0,Y 538.076,Z 314.958,A -85,B 0,C 180,E1 -3948.702,E2 -3948.702} C_VEL
LIN {X 0,Y 538.084,Z 314.954,A -85,B 0,C 180,E1 -3951.74,E2 -3951.74} C_VEL
LIN {X 0,Y 538.161,Z 314.95,A -85,B 0,C 180,E1 -3954.755,E2 -3954.755} C_VEL
LIN {X 0,Y 538.168,Z 314.943,A -85,B 0,C 180,E1 -3957.755,E2 -3957.755} C_VEL
LIN {X 0,Y 538.184,Z 314.95,A -85,B 0,C 180,E1 -3960.749,E2 -3960.749} C_VEL
LIN {X 0,Y 538.136,Z 314.953,A -85,B 0,C 180,E1 -3962.995,E2 -3962.995} C_VEL
LIN {X 0,Y 538.121,Z 314.95,A -85,B 0,C 180,E1 -3965.998,E2 -3965.998} C_VEL
LIN {X 0,Y 538.071,Z 314.959,A -85,B 0,C 180,E1 -3969.018,E2 -3969.018} C_VEL
LIN {X 0,Y 538.083,Z 314.957,A -85,B 0,C 180,E1 -3972.063,E2 -3972.063} C_VEL
LIN {X 0,Y 538.045,Z 314.959,A -85,B 0,C 180,E1 -3975.144,E2 -3975.144} C_VEL
LIN {X 0,Y 538.026,Z 314.969,A -85,B 0,C 180,E1 -3978.271,E2 -3978.271} C_VEL
LIN {X 0,Y 538.037,Z 314.964,A -85,B 0,C 180,E1 -3980.652,E2 -3980.652} C_VEL
LIN {X 0,Y 538.003,Z 314.968,A -85,B 0,C 180,E1 -3983.889,E2 -3983.889} C_VEL
LIN {X 0,Y 538.042,Z 314.965,A -85,B 0,C 180,E1 -3986.367,E2 -3986.367} C_VEL
LIN {X 0,Y 538.031,Z 314.961,A -85,B 0,C 180,E1 -3988.934,E2 -3988.934} C_VEL
LIN {X 0,Y 538.01,Z 314.97,A -85,B 0,C 180,E1 -3991.887,E2 -3991.887} C_VEL
LIN {X 0,Y 538.012,Z 314.964,A -85,B 0,C 180,E1 -3994.618,E2 -3994.618} C_VEL
LIN {X 0,Y 538.005,Z 314.966,A -85,B 0,C 180,E1 -3997.17,E2 -3997.17} C_VEL
LIN {X 0,Y 538.027,Z 314.97,A -85,B 0,C 180,E1 -3999.797,E2 -3999.797} C_VEL
LIN {X 0,Y 538.02,Z 314.966,A -85,B 0,C 180,E1 -4002.786,E2 -4002.786} C_VEL
LIN {X 0,Y 538.054,Z 315.258,A -85,B 0,C 180,E1 -4004.858,E2 -4004.858} C_VEL
LIN {X 0,Y 538.509,Z 318.608,A -85,B 0,C 180,E1 -4007.263,E2 -4007.263} C_VEL
LIN {X 0,Y 538.509,Z 321.659,A -85,B 0,C 180,E1 -4009.267,E2 -4009.267} C_VEL
LIN {X 0,Y 538.434,Z 326.351,A -85,B 0,C 180,E1 -4012.159,E2 -4012.159} C_VEL
LIN {X 0,Y 538.29,Z 331.179,A -85,B 0,C 180,E1 -4014.938,E2 -4014.938} C_VEL
LIN {X 0,Y 538.185,Z 336.128,A -85,B 0,C 180,E1 -4017.629,E2 -4017.629} C_VEL
LIN {X 0,Y 538.047,Z 341.197,A -85,B 0,C 180,E1 -4020.241,E2 -4020.241} C_VEL
LIN {X 0,Y 537.936,Z 346.347,A -85,B 0,C 180,E1 -4022.789,E2 -4022.789} C_VEL
LIN {X 0,Y 537.834,Z 351.579,A -85,B 0,C 180,E1 -4025.282,E2 -4025.282} C_VEL
LIN {X 0,Y 537.758,Z 358.606,A -85,B 0,C 180,E1 -4028.535,E2 -4028.535} C_VEL
LIN {X 0,Y 537.671,Z 364.052,A -85,B 0,C 180,E1 -4030.927,E2 -4030.927} C_VEL
LIN {X 0,Y 537.627,Z 369.525,A -85,B 0,C 180,E1 -4033.286,E2 -4033.286} C_VEL
LIN {X 0,Y 537.634,Z 374.986,A -85,B 0,C 180,E1 -4035.619,E2 -4035.619} C_VEL
LIN {X 0,Y 537.576,Z 377.485,A -85,B 0,C 180,E1 -4036.678,E2 -4036.678} C_VEL
LIN {X 0,Y 539.17,Z 387.881,A -85,B 0,C 180,E1 -4036.958,E2 -4036.958} C_VEL
LIN {X 0,Y 539.05,Z 396.986,A -85,B 0,C 180,E1 -4037.242,E2 -4037.242} C_VEL
LIN {X 0,Y 538.896,Z 406.342,A -85,B 0,C 180,E1 -4037.622,E2 -4037.622} C_VEL
LIN {X 0,Y 538.679,Z 416.815,A -85,B 0,C 180,E1 -4038.163,E2 -4038.163} C_VEL
LIN {X 0,Y 538.533,Z 425.443,A -85,B 0,C 180,E1 -4038.711,E2 -4038.711} C_VEL
LIN {X 0,Y 538.39,Z 434.148,A -85,B 0,C 180,E1 -4039.375,E2 -4039.375} C_VEL
LIN {X 0,Y 538.215,Z 441.52,A -85,B 0,C 180,E1 -4040.037,E2 -4040.037} C_VEL
LIN {X 0,Y 538.056,Z 448.713,A -85,B 0,C 180,E1 -4040.793,E2 -4040.793} C_VEL
LIN {X 0,Y 537.913,Z 454.89,A -85,B 0,C 180,E1 -4041.548,E2 -4041.548} C_VEL
LIN {X 0,Y 537.772,Z 461.398,A -85,B 0,C 180,E1 -4042.491,E2 -4042.491} C_VEL
LIN {X 0,Y 537.697,Z 466.65,A -85,B 0,C 180,E1 -4043.397,E2 -4043.397} C_VEL
LIN {X 0,Y 537.673,Z 471.336,A -85,B 0,C 180,E1 -4044.374,E2 -4044.374} C_VEL
LIN {X 0,Y 537.562,Z 475.63,A -85,B 0,C 180,E1 -4045.501,E2 -4045.501} C_VEL
LIN {X 0,Y 537.591,Z 477.974,A -85,B 0,C 180,E1 -4046.252,E2 -4046.252} C_VEL
LIN {X 0,Y 537.551,Z 479.763,A -85,B 0,C 180,E1 -4047.002,E2 -4047.002} C_VEL
LIN {X 0,Y 537.451,Z 482.19,A -85,B 0,C 180,E1 -4048.501,E2 -4048.501} C_VEL
LIN {X 0,Y 537.442,Z 482.773,A -85,B 0,C 180,E1 -4049.251,E2 -4049.251} C_VEL
LIN {X 0,Y 537.442,Z 482.773,A -85,B 0,C 180,E1 -4050.749,E2 -4050.749} C_VEL
LIN {X 0,Y 537.451,Z 482.19,A -85,B 0,C 180,E1 -4051.499,E2 -4051.499} C_VEL
LIN {X 0,Y 537.551,Z 479.763,A -85,B 0,C 180,E1 -4052.998,E2 -4052.998} C_VEL
LIN {X 0,Y 537.604,Z 476.839,A -85,B 0,C 180,E1 -4054.123,E2 -4054.123} C_VEL
LIN {X 0,Y 537.587,Z 472.88,A -85,B 0,C 180,E1 -4055.251,E2 -4055.251} C_VEL
LIN {X 0,Y 537.637,Z 468.088,A -85,B 0,C 180,E1 -4056.319,E2 -4056.319} C_VEL
LIN {X 0,Y 537.754,Z 462.548,A -85,B 0,C 180,E1 -4057.321,E2 -4057.321} C_VEL
LIN {X 0,Y 537.881,Z 456.26,A -85,B 0,C 180,E1 -4058.264,E2 -4058.264} C_VEL
LIN {X 0,Y 537.997,Z 450.334,A -85,B 0,C 180,E1 -4059.019,E2 -4059.019} C_VEL
LIN {X 0,Y 538.166,Z 443.433,A -85,B 0,C 180,E1 -4059.774,E2 -4059.774} C_VEL
LIN {X 0,Y 538.351,Z 435.28,A -85,B 0,C 180,E1 -4060.531,E2 -4060.531} C_VEL
LIN {X 0,Y 538.488,Z 426.792,A -85,B 0,C 180,E1 -4061.194,E2 -4061.194} C_VEL
LIN {X 0,Y 538.611,Z 418.378,A -85,B 0,C 180,E1 -4061.747,E2 -4061.747} C_VEL
LIN {X 0,Y 538.85,Z 408.353,A -85,B 0,C 180,E1 -4062.284,E2 -4062.284} C_VEL
LIN {X 0,Y 538.993,Z 399.562,A -85,B 0,C 180,E1 -4062.663,E2 -4062.663} C_VEL
LIN {X 0,Y 539.171,Z 389.63,A -85,B 0,C 180,E1 -4062.994,E2 -4062.994} C_VEL
LIN {X 0,Y 538.805,Z 384.809,A -85,B 0,C 180,E1 -4063.135,E2 -4063.135} C_VEL
LIN {X 0,Y 537.576,Z 377.485,A -85,B 0,C 180,E1 -4063.322,E2 -4063.322} C_VEL
LIN {X 0,Y 537.606,Z 371.346,A -85,B 0,C 180,E1 -4065.934,E2 -4065.934} C_VEL
LIN {X 0,Y 537.657,Z 365.877,A -85,B 0,C 180,E1 -4068.283,E2 -4068.283} C_VEL
LIN {X 0,Y 537.706,Z 360.397,A -85,B 0,C 180,E1 -4070.665,E2 -4070.665} C_VEL
LIN {X 0,Y 537.749,Z 355.099,A -85,B 0,C 180,E1 -4073.084,E2 -4073.084} C_VEL
LIN {X 0,Y 537.882,Z 349.618,A -85,B 0,C 180,E1 -4075.636,E2 -4075.636} C_VEL
LIN {X 0,Y 537.962,Z 344.597,A -85,B 0,C 180,E1 -4078.054,E2 -4078.054} C_VEL
LIN {X 0,Y 538.083,Z 339.484,A -85,B 0,C 180,E1 -4080.623,E2 -4080.623} C_VEL
LIN {X 0,Y 538.216,Z 334.357,A -85,B 0,C 180,E1 -4083.31,E2 -4083.31} C_VEL
LIN {X 0,Y 538.311,Z 329.537,A -85,B 0,C 180,E1 -4085.98,E2 -4085.98} C_VEL
LIN {X 0,Y 538.438,Z 324.749,A -85,B 0,C 180,E1 -4088.794,E2 -4088.794} C_VEL
LIN {X 0,Y 538.547,Z 320.109,A -85,B 0,C 180,E1 -4091.724,E2 -4091.724} C_VEL
LIN {X 0,Y 538.343,Z 317.125,A -85,B 0,C 180,E1 -4093.781,E2 -4093.781} C_VEL
LIN {X 0,Y 538.054,Z 315.254,A -85,B 0,C 180,E1 -4095.142,E2 -4095.142} C_VEL
LIN {X 0,Y 538.02,Z 314.966,A -85,B 0,C 180,E1 -4097.214,E2 -4097.214} C_VEL
LIN {X 0,Y 538.027,Z 314.97,A -85,B 0,C 180,E1 -4100.203,E2 -4100.203} C_VEL
LIN {X 0,Y 538.025,Z 314.963,A -85,B 0,C 180,E1 -4103.067,E2 -4103.067} C_VEL
LIN {X 0,Y 538.019,Z 314.97,A -85,B 0,C 180,E1 -4105.826,E2 -4105.826} C_VEL
LIN {X 0,Y 538.009,Z 314.965,A -85,B 0,C 180,E1 -4108.498,E2 -4108.498} C_VEL
LIN {X 0,Y 538.061,Z 314.957,A -85,B 0,C 180,E1 -4111.1,E2 -4111.1} C_VEL
LIN {X 0,Y 538.042,Z 314.965,A -85,B 0,C 180,E1 -4113.633,E2 -4113.633} C_VEL
LIN {X 0,Y 538.007,Z 314.967,A -85,B 0,C 180,E1 -4116.122,E2 -4116.122} C_VEL
LIN {X 0,Y 538.037,Z 314.964,A -85,B 0,C 180,E1 -4119.348,E2 -4119.348} C_VEL
LIN {X 0,Y 538.036,Z 314.96,A -85,B 0,C 180,E1 -4122.467,E2 -4122.467} C_VEL
LIN {X 0,Y 538.064,Z 314.964,A -85,B 0,C 180,E1 -4125.63,E2 -4125.63} C_VEL
LIN {X 0,Y 538.078,Z 314.955,A -85,B 0,C 180,E1 -4128.701,E2 -4128.701} C_VEL
LIN {X 0,Y 538.086,Z 314.957,A -85,B 0,C 180,E1 -4131.739,E2 -4131.739} C_VEL
LIN {X 0,Y 538.162,Z 314.946,A -85,B 0,C 180,E1 -4134.755,E2 -4134.755} C_VEL
LIN {X 0,Y 538.17,Z 314.945,A -85,B 0,C 180,E1 -4137.754,E2 -4137.754} C_VEL
LIN {X 0,Y 538.18,Z 314.945,A -85,B 0,C 180,E1 -4140.748,E2 -4140.748} C_VEL
LIN {X 0,Y 538.137,Z 314.955,A -85,B 0,C 180,E1 -4142.994,E2 -4142.994} C_VEL
LIN {X 0,Y 538.121,Z 314.949,A -85,B 0,C 180,E1 -4145.997,E2 -4145.997} C_VEL
LIN {X 0,Y 538.067,Z 314.964,A -85,B 0,C 180,E1 -4149.017,E2 -4149.017} C_VEL
LIN {X 0,Y 538.082,Z 314.954,A -85,B 0,C 180,E1 -4152.062,E2 -4152.062} C_VEL
LIN {X 0,Y 538.043,Z 314.963,A -85,B 0,C 180,E1 -4155.143,E2 -4155.143} C_VEL
LIN {X 0,Y 538.029,Z 314.963,A -85,B 0,C 180,E1 -4158.27,E2 -4158.27} C_VEL
LIN {X 0,Y 538.037,Z 314.969,A -85,B 0,C 180,E1 -4160.651,E2 -4160.651} C_VEL
LIN {X 0,Y 538.002,Z 314.965,A -85,B 0,C 180,E1 -4163.888,E2 -4163.888} C_VEL
LIN {X 0,Y 538.04,Z 314.966,A -85,B 0,C 180,E1 -4166.366,E2 -4166.366} C_VEL
LIN {X 0,Y 538.028,Z 314.964,A -85,B 0,C 180,E1 -4168.933,E2 -4168.933} C_VEL
LIN {X 0,Y 538.025,Z 314.963,A -85,B 0,C 180,E1 -4171.89,E2 -4171.89} C_VEL
LIN {X 0,Y 538.023,Z 314.966,A -85,B 0,C 180,E1 -4174.62,E2 -4174.62} C_VEL
LIN {X 0,Y 538.003,Z 314.964,A -85,B 0,C 180,E1 -4177.17,E2 -4177.17} C_VEL
LIN {X 0,Y 538.044,Z 314.959,A -85,B 0,C 180,E1 -4180.252,E2 -4180.252} C_VEL
LIN {X 0,Y 537.392,Z 315.042,A -85,B 0,C 180,E1 -4180.877,E2 -4180.877} C_VEL
LIN {X 0,Y 534.533,Z 315.401,A -85,B 0,C 180,E1 -4181.891,E2 -4181.891} C_VEL
LIN {X 0,Y 532.101,Z 315.703,A -85,B 0,C 180,E1 -4182.708,E2 -4182.708} C_VEL
LIN {X 0,Y 531.049,Z 315.832,A -85,B 0,C 180,E1 -4183.339,E2 -4183.339} C_VEL
LIN {X 0,Y 530.96,Z 315.842,A -85,B 0,C 180,E1 -4183.553,E2 -4183.553} C_VEL
LIN {X 0,Y 530.958,Z 315.844,A -85,B 0,C 180,E1 -4186.505,E2 -4186.505} C_VEL
LIN {X 0,Y 531.023,Z 315.837,A -85,B 0,C 180,E1 -4189.571,E2 -4189.571} C_VEL
LIN {X 0,Y 530.965,Z 315.841,A -85,B 0,C 180,E1 -4192.577,E2 -4192.577} C_VEL
LIN {X 0,Y 530.992,Z 315.839,A -85,B 0,C 180,E1 -4195.311,E2 -4195.311} C_VEL
LIN {X 0,Y 530.98,Z 315.844,A -85,B 0,C 180,E1 -4198.033,E2 -4198.033} C_VEL
LIN {X 0,Y 530.986,Z 315.838,A -85,B 0,C 180,E1 -4200.874,E2 -4200.874} C_VEL
LIN {X 0,Y 531.009,Z 315.839,A -85,B 0,C 180,E1 -4203.257,E2 -4203.257} C_VEL
LIN {X 0,Y 530.982,Z 315.842,A -85,B 0,C 180,E1 -4205.96,E2 -4205.96} C_VEL
LIN {X 0,Y 530.997,Z 315.839,A -85,B 0,C 180,E1 -4209.062,E2 -4209.062} C_VEL
LIN {X 0,Y 531.013,Z 315.836,A -85,B 0,C 180,E1 -4212.278,E2 -4212.278} C_VEL
LIN {X 0,Y 531.037,Z 315.84,A -85,B 0,C 180,E1 -4215.436,E2 -4215.436} C_VEL
LIN {X 0,Y 531.034,Z 315.834,A -85,B 0,C 180,E1 -4218.55,E2 -4218.55} C_VEL
LIN {X 0,Y 531.054,Z 315.835,A -85,B 0,C 180,E1 -4221.629,E2 -4221.629} C_VEL
LIN {X 0,Y 531.122,Z 315.826,A -85,B 0,C 180,E1 -4224.685,E2 -4224.685} C_VEL
LIN {X 0,Y 531.139,Z 315.821,A -85,B 0,C 180,E1 -4227.725,E2 -4227.725} C_VEL
LIN {X 0,Y 531.15,Z 315.825,A -85,B 0,C 180,E1 -4230.758,E2 -4230.758} C_VEL
LIN {X 0,Y 531.102,Z 315.832,A -85,B 0,C 180,E1 -4233.034,E2 -4233.034} C_VEL
LIN {X 0,Y 531.089,Z 315.827,A -85,B 0,C 180,E1 -4236.077,E2 -4236.077} C_VEL
LIN {X 0,Y 531.029,Z 315.839,A -85,B 0,C 180,E1 -4239.138,E2 -4239.138} C_VEL
LIN {X 0,Y 531.038,Z 315.835,A -85,B 0,C 180,E1 -4242.225,E2 -4242.225} C_VEL
LIN {X 0,Y 530.992,Z 315.84,A -85,B 0,C 180,E1 -4245.35,E2 -4245.35} C_VEL
LIN {X 0,Y 530.988,Z 315.847,A -85,B 0,C 180,E1 -4248.521,E2 -4248.521} C_VEL
LIN {X 0,Y 530.997,Z 315.839,A -85,B 0,C 180,E1 -4250.938,E2 -4250.938} C_VEL
LIN {X 0,Y 530.969,Z 315.846,A -85,B 0,C 180,E1 -4254.225,E2 -4254.225} C_VEL
LIN {X 0,Y 531.009,Z 315.839,A -85,B 0,C 180,E1 -4256.743,E2 -4256.743} C_VEL
LIN {X 0,Y 530.979,Z 315.839,A -85,B 0,C 180,E1 -4259.323,E2 -4259.323} C_VEL
LIN {X 0,Y 530.977,Z 315.846,A -85,B 0,C 180,E1 -4262.103,E2 -4262.103} C_VEL
LIN {X 0,Y 530.979,Z 315.84,A -85,B 0,C 180,E1 -4264.853,E2 -4264.853} C_VEL
LIN {X 0,Y 530.963,Z 315.842,A -85,B 0,C 180,E1 -4267.508,E2 -4267.508} C_VEL
LIN {X 0,Y 531.023,Z 315.837,A -85,B 0,C 180,E1 -4270.429,E2 -4270.429} C_VEL
LIN {X 0,Y 530.958,Z 315.844,A -85,B 0,C 180,E1 -4273.495,E2 -4273.495} C_VEL
LIN {X 0,Y 530.963,Z 315.842,A -85,B 0,C 180,E1 -4276.506,E2 -4276.506} C_VEL
LIN {X 0,Y 531.023,Z 315.839,A -85,B 0,C 180,E1 -4279.572,E2 -4279.572} C_VEL
LIN {X 0,Y 530.965,Z 315.841,A -85,B 0,C 180,E1 -4282.577,E2 -4282.577} C_VEL
LIN {X 0,Y 530.979,Z 315.843,A -85,B 0,C 180,E1 -4285.31,E2 -4285.31} C_VEL
LIN {X 0,Y 530.98,Z 315.842,A -85,B 0,C 180,E1 -4288.033,E2 -4288.033} C_VEL
LIN {X 0,Y 530.986,Z 315.839,A -85,B 0,C 180,E1 -4290.874,E2 -4290.874} C_VEL
LIN {X 0,Y 531.002,Z 315.842,A -85,B 0,C 180,E1 -4293.257,E2 -4293.257} C_VEL
LIN {X 0,Y 530.983,Z 315.84,A -85,B 0,C 180,E1 -4295.961,E2 -4295.961} C_VEL
LIN {X 0,Y 530.998,Z 315.842,A -85,B 0,C 180,E1 -4299.063,E2 -4299.063} C_VEL
LIN {X 0,Y 531.015,Z 315.834,A -85,B 0,C 180,E1 -4302.278,E2 -4302.278} C_VEL
LIN {X 0,Y 531.017,Z 315.839,A -85,B 0,C 180,E1 -4305.436,E2 -4305.436} C_VEL
LIN {X 0,Y 531.035,Z 315.834,A -85,B 0,C 180,E1 -4308.55,E2 -4308.55} C_VEL
LIN {X 0,Y 531.054,Z 315.831,A -85,B 0,C 180,E1 -4311.63,E2 -4311.63} C_VEL
LIN {X 0,Y 531.12,Z 315.826,A -85,B 0,C 180,E1 -4314.686,E2 -4314.686} C_VEL
LIN {X 0,Y 531.14,Z 315.819,A -85,B 0,C 180,E1 -4317.725,E2 -4317.725} C_VEL
LIN {X 0,Y 531.153,Z 315.826,A -85,B 0,C 180,E1 -4320.759,E2 -4320.759} C_VEL
LIN {X 0,Y 531.103,Z 315.828,A -85,B 0,C 180,E1 -4323.035,E2 -4323.035} C_VEL
LIN {X 0,Y 531.076,Z 315.828,A -85,B 0,C 180,E1 -4326.078,E2 -4326.078} C_VEL
LIN {X 0,Y 531.055,Z 315.835,A -85,B 0,C 180,E1 -4328.371,E2 -4328.371} C_VEL
LIN {X 0,Y 531.052,Z 315.83,A -85,B 0,C 180,E1 -4331.673,E2 -4331.673} C_VEL
LIN {X 0,Y 531.031,Z 315.835,A -85,B 0,C 180,E1 -4334.956,E2 -4334.956} C_VEL
LIN {X 0,Y 530.981,Z 315.84,A -85,B 0,C 180,E1 -4337.724,E2 -4337.724} C_VEL
LIN {X 0,Y 531.025,Z 315.839,A -85,B 0,C 180,E1 -4340.128,E2 -4340.128} C_VEL
LIN {X 0,Y 530.945,Z 315.848,A -85,B 0,C 180,E1 -4342.574,E2 -4342.574} C_VEL
LIN {X 0,Y 530.995,Z 315.837,A -85,B 0,C 180,E1 -4345.058,E2 -4345.058} C_VEL
LIN {X 0,Y 531.014,Z 315.836,A -85,B 0,C 180,E1 -4347.596,E2 -4347.596} C_VEL
LIN {X 0,Y 530.974,Z 315.841,A -85,B 0,C 180,E1 -4350.645,E2 -4350.645} C_VEL
LIN {X 0,Y 530.988,Z 315.843,A -85,B 0,C 180,E1 -4353.773,E2 -4353.773} C_VEL
LIN {X 0,Y 530.956,Z 315.845,A -85,B 0,C 180,E1 -4356.559,E2 -4356.559} C_VEL
LIN {X 0,Y 530.989,Z 315.843,A -85,B 0,C 180,E1 -4359.444,E2 -4359.444} C_VEL
LIN {X 0,Y 530.979,Z 315.845,A -85,B 0,C 180,E1 -4362.457,E2 -4362.457} C_VEL
LIN {X 0,Y 530.99,Z 315.866,A -85,B 0,C 180,E1 -4364.38,E2 -4364.38} C_VEL
LIN {X 0,Y 531.422,Z 318.961,A -85,B 0,C 180,E1 -4366.667,E2 -4366.667} C_VEL
LIN {X 0,Y 531.522,Z 322.258,A -85,B 0,C 180,E1 -4368.91,E2 -4368.91} C_VEL
LIN {X 0,Y 531.427,Z 326.476,A -85,B 0,C 180,E1 -4371.57,E2 -4371.57} C_VEL
LIN {X 0,Y 531.3,Z 331.267,A -85,B 0,C 180,E1 -4374.407,E2 -4374.407} C_VEL
LIN {X 0,Y 531.162,Z 336.189,A -85,B 0,C 180,E1 -4377.147,E2 -4377.147} C_VEL
LIN {X 0,Y 531.013,Z 341.218,A -85,B 0,C 180,E1 -4379.806,E2 -4379.806} C_VEL
LIN {X 0,Y 530.892,Z 346.548,A -85,B 0,C 180,E1 -4382.493,E2 -4382.493} C_VEL
LIN {X 0,Y 530.771,Z 351.555,A -85,B 0,C 180,E1 -4384.931,E2 -4384.931} C_VEL
LIN {X 0,Y 530.689,Z 358.599,A -85,B 0,C 180,E1 -4388.235,E2 -4388.235} C_VEL
LIN {X 0,Y 530.628,Z 363.96,A -85,B 0,C 180,E1 -4390.663,E2 -4390.663} C_VEL
LIN {X 0,Y 530.541,Z 369.433,A -85,B 0,C 180,E1 -4393.056,E2 -4393.056} C_VEL
LIN {X 0,Y 530.548,Z 374.895,A -85,B 0,C 180,E1 -4395.423,E2 -4395.423} C_VEL
LIN {X 0,Y 530.49,Z 377.524,A -85,B 0,C 180,E1 -4396.509,E2 -4396.509} C_VEL
LIN {X 0,Y 532.193,Z 387.683,A -85,B 0,C 180,E1 -4396.784,E2 -4396.784} C_VEL
LIN {X 0,Y 532.132,Z 396.79,A -85,B 0,C 180,E1 -4397.074,E2 -4397.074} C_VEL
LIN {X 0,Y 531.916,Z 407.156,A -85,B 0,C 180,E1 -4397.505,E2 -4397.505} C_VEL
LIN {X 0,Y 531.7,Z 416.505,A -85,B 0,C 180,E1 -4397.997,E2 -4397.997} C_VEL
LIN {X 0,Y 531.554,Z 425.297,A -85,B 0,C 180,E1 -4398.561,E2 -4398.561} C_VEL
LIN {X 0,Y 531.362,Z 434.029,A -85,B 0,C 180,E1 -4399.233,E2 -4399.233} C_VEL
LIN {X 0,Y 531.173,Z 441.427,A -85,B 0,C 180,E1 -4399.903,E2 -4399.903} C_VEL
LIN {X 0,Y 531.004,Z 448.649,A -85,B 0,C 180,E1 -4400.669,E2 -4400.669} C_VEL
LIN {X 0,Y 530.879,Z 454.852,A -85,B 0,C 180,E1 -4401.435,E2 -4401.435} C_VEL
LIN {X 0,Y 530.706,Z 461.387,A -85,B 0,C 180,E1 -4402.39,E2 -4402.39} C_VEL
LIN {X 0,Y 530.596,Z 467.204,A -85,B 0,C 180,E1 -4403.421,E2 -4403.421} C_VEL
LIN {X 0,Y 530.607,Z 471.328,A -85,B 0,C 180,E1 -4404.299,E2 -4404.299} C_VEL
LIN {X 0,Y 530.462,Z 475.624,A -85,B 0,C 180,E1 -4405.441,E2 -4405.441} C_VEL
LIN {X 0,Y 530.516,Z 477.972,A -85,B 0,C 180,E1 -4406.202,E2 -4406.202} C_VEL
LIN {X 0,Y 530.457,Z 479.757,A -85,B 0,C 180,E1 -4406.962,E2 -4406.962} C_VEL
LIN {X 0,Y 530.361,Z 482.182,A -85,B 0,C 180,E1 -4408.481,E2 -4408.481} C_VEL
LIN {X 0,Y 530.344,Z 482.766,A -85,B 0,C 180,E1 -4409.241,E2 -4409.241} C_VEL
LIN {X 0,Y 530.344,Z 482.766,A -85,B 0,C 180,E1 -4410.759,E2 -4410.759} C_VEL
LIN {X 0,Y 530.361,Z 482.182,A -85,B 0,C 180,E1 -4411.519,E2 -4411.519} C_VEL
LIN {X 0,Y 530.457,Z 479.757,A -85,B 0,C 180,E1 -4413.038,E2 -4413.038} C_VEL
LIN {X 0,Y 530.524,Z 476.832,A -85,B 0,C 180,E1 -4414.178,E2 -4414.178} C_VEL
LIN {X 0,Y 530.523,Z 472.872,A -85,B 0,C 180,E1 -4415.321,E2 -4415.321} C_VEL
LIN {X 0,Y 530.551,Z 468.572,A -85,B 0,C 180,E1 -4416.305,E2 -4416.305} C_VEL
LIN {X 0,Y 530.666,Z 463.69,A -85,B 0,C 180,E1 -4417.228,E2 -4417.228} C_VEL
LIN {X 0,Y 530.812,Z 457.604,A -85,B 0,C 180,E1 -4418.183,E2 -4418.183} C_VEL
LIN {X 0,Y 530.918,Z 451.903,A -85,B 0,C 180,E1 -4418.948,E2 -4418.948} C_VEL
LIN {X 0,Y 531.127,Z 443.347,A -85,B 0,C 180,E1 -4419.905,E2 -4419.905} C_VEL
LIN {X 0,Y 531.35,Z 435.165,A -85,B 0,C 180,E1 -4420.671,E2 -4420.671} C_VEL
LIN {X 0,Y 531.509,Z 426.648,A -85,B 0,C 180,E1 -4421.343,E2 -4421.343} C_VEL
LIN {X 0,Y 531.661,Z 417.914,A -85,B 0,C 180,E1 -4421.921,E2 -4421.921} C_VEL
LIN {X 0,Y 531.899,Z 408.164,A -85,B 0,C 180,E1 -4422.447,E2 -4422.447} C_VEL
LIN {X 0,Y 532.044,Z 399.365,A -85,B 0,C 180,E1 -4422.831,E2 -4422.831} C_VEL
LIN {X 0,Y 532.273,Z 389.435,A -85,B 0,C 180,E1 -4423.165,E2 -4423.165} C_VEL
LIN {X 0,Y 530.987,Z 380.537,A -85,B 0,C 180,E1 -4423.423,E2 -4423.423} C_VEL
LIN {X 0,Y 530.469,Z 377.365,A -85,B 0,C 180,E1 -4423.504,E2 -4423.504} C_VEL
LIN {X 0,Y 530.514,Z 371.255,A -85,B 0,C 180,E1 -4426.153,E2 -4426.153} C_VEL
LIN {X 0,Y 530.574,Z 365.785,A -85,B 0,C 180,E1 -4428.536,E2 -4428.536} C_VEL
LIN {X 0,Y 530.647,Z 360.357,A -85,B 0,C 180,E1 -4430.952,E2 -4430.952} C_VEL
LIN {X 0,Y 530.72,Z 353.848,A -85,B 0,C 180,E1 -4433.974,E2 -4433.974} C_VEL
LIN {X 0,Y 530.86,Z 348.045,A -85,B 0,C 180,E1 -4436.751,E2 -4436.751} C_VEL
LIN {X 0,Y 530.979,Z 342.911,A -85,B 0,C 180,E1 -4439.323,E2 -4439.323} C_VEL
LIN {X 0,Y 531.108,Z 337.52,A -85,B 0,C 180,E1 -4442.124,E2 -4442.124} C_VEL
LIN {X 0,Y 531.268,Z 332.485,A -85,B 0,C 180,E1 -4444.897,E2 -4444.897} C_VEL
LIN {X 0,Y 531.372,Z 328.027,A -85,B 0,C 180,E1 -4447.479,E2 -4447.479} C_VEL
LIN {X 0,Y 531.499,Z 323.339,A -85,B 0,C 180,E1 -4450.385,E2 -4450.385} C_VEL
LIN {X 0,Y 531.53,Z 320.285,A -85,B 0,C 180,E1 -4452.402,E2 -4452.402} C_VEL
LIN {X 0,Y 531.181,Z 317.325,A -85,B 0,C 180,E1 -4454.526,E2 -4454.526} C_VEL
LIN {X 0,Y 530.99,Z 315.867,A -85,B 0,C 180,E1 -4455.62,E2 -4455.62} C_VEL
LIN {X 0,Y 530.994,Z 315.844,A -85,B 0,C 180,E1 -4458.564,E2 -4458.564} C_VEL
LIN {X 0,Y 530.959,Z 315.846,A -85,B 0,C 180,E1 -4461.529,E2 -4461.529} C_VEL
LIN {X 0,Y 530.955,Z 315.848,A -85,B 0,C 180,E1 -4464.38,E2 -4464.38} C_VEL
LIN {X 0,Y 530.967,Z 315.84,A -85,B 0,C 180,E1 -4467.133,E2 -4467.133} C_VEL
LIN {X 0,Y 530.97,Z 315.847,A -85,B 0,C 180,E1 -4469.803,E2 -4469.803} C_VEL
LIN {X 0,Y 531.013,Z 315.836,A -85,B 0,C 180,E1 -4472.467,E2 -4472.467} C_VEL
LIN {X 0,Y 530.995,Z 315.837,A -85,B 0,C 180,E1 -4474.942,E2 -4474.942} C_VEL
LIN {X 0,Y 530.971,Z 315.842,A -85,B 0,C 180,E1 -4478.246,E2 -4478.246} C_VEL
LIN {X 0,Y 530.992,Z 315.837,A -85,B 0,C 180,E1 -4480.677,E2 -4480.677} C_VEL
LIN {X 0,Y 530.975,Z 315.841,A -85,B 0,C 180,E1 -4483.07,E2 -4483.07} C_VEL
LIN {X 0,Y 531.041,Z 315.839,A -85,B 0,C 180,E1 -4485.436,E2 -4485.436} C_VEL
LIN {X 0,Y 531.037,Z 315.832,A -85,B 0,C 180,E1 -4488.549,E2 -4488.549} C_VEL
LIN {X 0,Y 531.055,Z 315.835,A -85,B 0,C 180,E1 -4491.629,E2 -4491.629} C_VEL
LIN {X 0,Y 531.121,Z 315.822,A -85,B 0,C 180,E1 -4494.685,E2 -4494.685} C_VEL
LIN {X 0,Y 531.141,Z 315.821,A -85,B 0,C 180,E1 -4497.725,E2 -4497.725} C_VEL
LIN {X 0,Y 531.15,Z 315.821,A -85,B 0,C 180,E1 -4500.758,E2 -4500.758} C_VEL
LIN {X 0,Y 531.104,Z 315.831,A -85,B 0,C 180,E1 -4503.034,E2 -4503.034} C_VEL
LIN {X 0,Y 531.076,Z 315.827,A -85,B 0,C 180,E1 -4506.077,E2 -4506.077} C_VEL
LIN {X 0,Y 531.054,Z 315.831,A -85,B 0,C 180,E1 -4508.37,E2 -4508.37} C_VEL
LIN {X 0,Y 531.05,Z 315.83,A -85,B 0,C 180,E1 -4511.672,E2 -4511.672} C_VEL
LIN {X 0,Y 531.029,Z 315.84,A -85,B 0,C 180,E1 -4514.955,E2 -4514.955} C_VEL
LIN {X 0,Y 531.015,Z 315.834,A -85,B 0,C 180,E1 -4517.722,E2 -4517.722} C_VEL
LIN {X 0,Y 530.998,Z 315.842,A -85,B 0,C 180,E1 -4520.937,E2 -4520.937} C_VEL
LIN {X 0,Y 530.969,Z 315.844,A -85,B 0,C 180,E1 -4524.224,E2 -4524.224} C_VEL
LIN {X 0,Y 531.002,Z 315.842,A -85,B 0,C 180,E1 -4526.743,E2 -4526.743} C_VEL
LIN {X 0,Y 530.979,Z 315.839,A -85,B 0,C 180,E1 -4529.322,E2 -4529.322} C_VEL
LIN {X 0,Y 530.978,Z 315.844,A -85,B 0,C 180,E1 -4532.103,E2 -4532.103} C_VEL
LIN {X 0,Y 530.98,Z 315.841,A -85,B 0,C 180,E1 -4534.853,E2 -4534.853} C_VEL
LIN {X 0,Y 530.963,Z 315.841,A -85,B 0,C 180,E1 -4537.507,E2 -4537.507} C_VEL
LIN {X 0,Y 531.023,Z 315.839,A -85,B 0,C 180,E1 -4540.428,E2 -4540.428} C_VEL
LIN {X 0,Y 530.96,Z 315.842,A -85,B 0,C 180,E1 -4543.553,E2 -4543.553} C_VEL
LIN {X 0,Y 530.286,Z 315.933,A -85,B 0,C 180,E1 -4544.186,E2 -4544.186} C_VEL
LIN {X 0,Y 527.437,Z 316.281,A -85,B 0,C 180,E1 -4545.215,E2 -4545.215} C_VEL
LIN {X 0,Y 525.033,Z 316.589,A -85,B 0,C 180,E1 -4546.043,E2 -4546.043} C_VEL
LIN {X 0,Y 524.001,Z 316.71,A -85,B 0,C 180,E1 -4546.683,E2 -4546.683} C_VEL
LIN {X 0,Y 523.916,Z 316.719,A -85,B 0,C 180,E1 -4546.899,E2 -4546.899} C_VEL
LIN {X 0,Y 523.975,Z 316.72,A -85,B 0,C 180,E1 -4549.923,E2 -4549.923} C_VEL
LIN {X 0,Y 523.907,Z 316.72,A -85,B 0,C 180,E1 -4552.868,E2 -4552.868} C_VEL
LIN {X 0,Y 523.937,Z 316.723,A -85,B 0,C 180,E1 -4555.71,E2 -4555.71} C_VEL
LIN {X 0,Y 523.928,Z 316.718,A -85,B 0,C 180,E1 -4558.457,E2 -4558.457} C_VEL
LIN {X 0,Y 523.937,Z 316.718,A -85,B 0,C 180,E1 -4561.125,E2 -4561.125} C_VEL
LIN {X 0,Y 523.983,Z 316.714,A -85,B 0,C 180,E1 -4563.98,E2 -4563.98} C_VEL
LIN {X 0,Y 523.922,Z 316.719,A -85,B 0,C 180,E1 -4566.27,E2 -4566.27} C_VEL
LIN {X 0,Y 523.943,Z 316.716,A -85,B 0,C 180,E1 -4568.767,E2 -4568.767} C_VEL
LIN {X 0,Y 523.949,Z 316.721,A -85,B 0,C 180,E1 -4571.221,E2 -4571.221} C_VEL
LIN {X 0,Y 523.934,Z 316.724,A -85,B 0,C 180,E1 -4573.639,E2 -4573.639} C_VEL
LIN {X 0,Y 523.942,Z 316.718,A -85,B 0,C 180,E1 -4576.028,E2 -4576.028} C_VEL
LIN {X 0,Y 524.009,Z 316.708,A -85,B 0,C 180,E1 -4578.394,E2 -4578.394} C_VEL
LIN {X 0,Y 524.002,Z 316.714,A -85,B 0,C 180,E1 -4581.516,E2 -4581.516} C_VEL
LIN {X 0,Y 524.084,Z 316.702,A -85,B 0,C 180,E1 -4584.614,E2 -4584.614} C_VEL
LIN {X 0,Y 524.111,Z 316.697,A -85,B 0,C 180,E1 -4587.694,E2 -4587.694} C_VEL
LIN {X 0,Y 524.121,Z 316.701,A -85,B 0,C 180,E1 -4590.768,E2 -4590.768} C_VEL
LIN {X 0,Y 524.069,Z 316.708,A -85,B 0,C 180,E1 -4593.075,E2 -4593.075} C_VEL
LIN {X 0,Y 524.05,Z 316.705,A -85,B 0,C 180,E1 -4596.159,E2 -4596.159} C_VEL
LIN {X 0,Y 523.997,Z 316.713,A -85,B 0,C 180,E1 -4599.262,E2 -4599.262} C_VEL
LIN {X 0,Y 524,Z 316.709,A -85,B 0,C 180,E1 -4601.74,E2 -4601.74} C_VEL
LIN {X 0,Y 523.991,Z 316.714,A -85,B 0,C 180,E1 -4605.053,E2 -4605.053} C_VEL
LIN {X 0,Y 523.961,Z 316.716,A -85,B 0,C 180,E1 -4607.969,E2 -4607.969} C_VEL
LIN {X 0,Y 523.969,Z 316.72,A -85,B 0,C 180,E1 -4610.41,E2 -4610.41} C_VEL
LIN {X 0,Y 523.908,Z 316.723,A -85,B 0,C 180,E1 -4612.894,E2 -4612.894} C_VEL
LIN {X 0,Y 523.951,Z 316.714,A -85,B 0,C 180,E1 -4615.419,E2 -4615.419} C_VEL
LIN {X 0,Y 523.968,Z 316.716,A -85,B 0,C 180,E1 -4617.999,E2 -4617.999} C_VEL
LIN {X 0,Y 523.944,Z 316.717,A -85,B 0,C 180,E1 -4620.855,E2 -4620.855} C_VEL
LIN {X 0,Y 523.957,Z 316.716,A -85,B 0,C 180,E1 -4623.735,E2 -4623.735} C_VEL
LIN {X 0,Y 523.916,Z 316.723,A -85,B 0,C 180,E1 -4626.404,E2 -4626.404} C_VEL
LIN {X 0,Y 523.929,Z 316.717,A -85,B 0,C 180,E1 -4629.084,E2 -4629.084} C_VEL
LIN {X 0,Y 523.954,Z 316.721,A -85,B 0,C 180,E1 -4632.119,E2 -4632.119} C_VEL
LIN {X 0,Y 523.953,Z 316.716,A -85,B 0,C 180,E1 -4635.309,E2 -4635.309} C_VEL
LIN {X 0,Y 523.969,Z 316.712,A -85,B 0,C 180,E1 -4638.688,E2 -4638.688} C_VEL
LIN {X 0,Y 523.922,Z 316.719,A -85,B 0,C 180,E1 -4641.08,E2 -4641.08} C_VEL
LIN {X 0,Y 523.897,Z 316.728,A -85,B 0,C 180,E1 -4643.826,E2 -4643.826} C_VEL
LIN {X 0,Y 523.939,Z 316.716,A -85,B 0,C 180,E1 -4646.636,E2 -4646.636} C_VEL
LIN {X 0,Y 523.954,Z 316.72,A -85,B 0,C 180,E1 -4649.356,E2 -4649.356} C_VEL
LIN {X 0,Y 523.976,Z 316.712,A -85,B 0,C 180,E1 -4652.281,E2 -4652.281} C_VEL
LIN {X 0,Y 523.95,Z 316.715,A -85,B 0,C 180,E1 -4654.582,E2 -4654.582} C_VEL
LIN {X 0,Y 523.909,Z 316.725,A -85,B 0,C 180,E1 -4657.107,E2 -4657.107} C_VEL
LIN {X 0,Y 523.977,Z 316.713,A -85,B 0,C 180,E1 -4659.866,E2 -4659.866} C_VEL
LIN {X 0,Y 523.965,Z 316.716,A -85,B 0,C 180,E1 -4662.838,E2 -4662.838} C_VEL
LIN {X 0,Y 523.975,Z 316.72,A -85,B 0,C 180,E1 -4665.236,E2 -4665.236} C_VEL
LIN {X 0,Y 524.011,Z 316.708,A -85,B 0,C 180,E1 -4668.395,E2 -4668.395} C_VEL
LIN {X 0,Y 524.002,Z 316.71,A -85,B 0,C 180,E1 -4671.516,E2 -4671.516} C_VEL
LIN {X 0,Y 524.081,Z 316.702,A -85,B 0,C 180,E1 -4674.614,E2 -4674.614} C_VEL
LIN {X 0,Y 524.112,Z 316.694,A -85,B 0,C 180,E1 -4677.695,E2 -4677.695} C_VEL
LIN {X 0,Y 524.123,Z 316.702,A -85,B 0,C 180,E1 -4680.769,E2 -4680.769} C_VEL
LIN {X 0,Y 524.07,Z 316.704,A -85,B 0,C 180,E1 -4683.075,E2 -4683.075} C_VEL
LIN {X 0,Y 524.037,Z 316.706,A -85,B 0,C 180,E1 -4686.16,E2 -4686.16} C_VEL
LIN {X 0,Y 524.004,Z 316.715,A -85,B 0,C 180,E1 -4688.484,E2 -4688.484} C_VEL
LIN {X 0,Y 524.003,Z 316.708,A -85,B 0,C 180,E1 -4691.74,E2 -4691.74} C_VEL
LIN {X 0,Y 523.994,Z 316.71,A -85,B 0,C 180,E1 -4695.053,E2 -4695.053} C_VEL
LIN {X 0,Y 523.947,Z 316.718,A -85,B 0,C 180,E1 -4697.97,E2 -4697.97} C_VEL
LIN {X 0,Y 523.972,Z 316.72,A -85,B 0,C 180,E1 -4700.41,E2 -4700.41} C_VEL
LIN {X 0,Y 523.911,Z 316.721,A -85,B 0,C 180,E1 -4702.894,E2 -4702.894} C_VEL
LIN {X 0,Y 523.985,Z 316.717,A -85,B 0,C 180,E1 -4706.02,E2 -4706.02} C_VEL
LIN {X 0,Y 523.939,Z 316.716,A -85,B 0,C 180,E1 -4708.875,E2 -4708.875} C_VEL
LIN {X 0,Y 523.921,Z 316.72,A -85,B 0,C 180,E1 -4711.545,E2 -4711.545} C_VEL
LIN {X 0,Y 523.933,Z 316.722,A -85,B 0,C 180,E1 -4714.291,E2 -4714.291} C_VEL
LIN {X 0,Y 523.908,Z 316.722,A -85,B 0,C 180,E1 -4717.133,E2 -4717.133} C_VEL
LIN {X 0,Y 523.939,Z 316.724,A -85,B 0,C 180,E1 -4720.13,E2 -4720.13} C_VEL
LIN {X 0,Y 523.936,Z 316.723,A -85,B 0,C 180,E1 -4722.459,E2 -4722.459} C_VEL
LIN {X 0,Y 523.962,Z 316.898,A -85,B 0,C 180,E1 -4724.226,E2 -4724.226} C_VEL
LIN {X 0,Y 524.438,Z 320.483,A -85,B 0,C 180,E1 -4726.886,E2 -4726.886} C_VEL
LIN {X 0,Y 524.525,Z 323.49,A -85,B 0,C 180,E1 -4728.964,E2 -4728.964} C_VEL
LIN {X 0,Y 524.414,Z 328.176,A -85,B 0,C 180,E1 -4731.941,E2 -4731.941} C_VEL
LIN {X 0,Y 524.265,Z 333.076,A -85,B 0,C 180,E1 -4734.859,E2 -4734.859} C_VEL
LIN {X 0,Y 524.104,Z 338.09,A -85,B 0,C 180,E1 -4737.651,E2 -4737.651} C_VEL
LIN {X 0,Y 523.956,Z 343.772,A -85,B 0,C 180,E1 -4740.677,E2 -4740.677} C_VEL
LIN {X 0,Y 523.777,Z 349.79,A -85,B 0,C 180,E1 -4743.718,E2 -4743.718} C_VEL
LIN {X 0,Y 523.649,Z 355.023,A -85,B 0,C 180,E1 -4746.257,E2 -4746.257} C_VEL
LIN {X 0,Y 523.574,Z 360.309,A -85,B 0,C 180,E1 -4748.751,E2 -4748.751} C_VEL
LIN {X 0,Y 523.515,Z 365.676,A -85,B 0,C 180,E1 -4751.205,E2 -4751.205} C_VEL
LIN {X 0,Y 523.424,Z 371.102,A -85,B 0,C 180,E1 -4753.622,E2 -4753.622} C_VEL
LIN {X 0,Y 523.412,Z 377.179,A -85,B 0,C 180,E1 -4756.311,E2 -4756.311} C_VEL
LIN {X 0,Y 525.325,Z 389.238,A -85,B 0,C 180,E1 -4756.657,E2 -4756.657} C_VEL
LIN {X 0,Y 525.095,Z 401.744,A -85,B 0,C 180,E1 -4757.094,E2 -4757.094} C_VEL
LIN {X 0,Y 524.838,Z 413.915,A -85,B 0,C 180,E1 -4757.693,E2 -4757.693} C_VEL
LIN {X 0,Y 524.59,Z 423.796,A -85,B 0,C 180,E1 -4758.313,E2 -4758.313} C_VEL
LIN {X 0,Y 524.38,Z 432.697,A -85,B 0,C 180,E1 -4758.99,E2 -4758.99} C_VEL
LIN {X 0,Y 524.153,Z 441.23,A -85,B 0,C 180,E1 -4759.767,E2 -4759.767} C_VEL
LIN {X 0,Y 523.98,Z 448.452,A -85,B 0,C 180,E1 -4760.543,E2 -4760.543} C_VEL
LIN {X 0,Y 523.809,Z 454.655,A -85,B 0,C 180,E1 -4761.318,E2 -4761.318} C_VEL
LIN {X 0,Y 523.659,Z 461.192,A -85,B 0,C 180,E1 -4762.287,E2 -4762.287} C_VEL
LIN {X 0,Y 523.575,Z 465.694,A -85,B 0,C 180,E1 -4763.061,E2 -4763.061} C_VEL
LIN {X 0,Y 523.519,Z 471.183,A -85,B 0,C 180,E1 -4764.221,E2 -4764.221} C_VEL
LIN {X 0,Y 523.366,Z 475.501,A -85,B 0,C 180,E1 -4765.379,E2 -4765.379} C_VEL
LIN {X 0,Y 523.444,Z 477.867,A -85,B 0,C 180,E1 -4766.151,E2 -4766.151} C_VEL
LIN {X 0,Y 523.368,Z 479.66,A -85,B 0,C 180,E1 -4766.921,E2 -4766.921} C_VEL
LIN {X 0,Y 523.275,Z 482.098,A -85,B 0,C 180,E1 -4768.461,E2 -4768.461} C_VEL
LIN {X 0,Y 523.25,Z 482.684,A -85,B 0,C 180,E1 -4769.23,E2 -4769.23} C_VEL
LIN {X 0,Y 523.25,Z 482.684,A -85,B 0,C 180,E1 -4770.77,E2 -4770.77} C_VEL
LIN {X 0,Y 523.275,Z 482.098,A -85,B 0,C 180,E1 -4771.539,E2 -4771.539} C_VEL
LIN {X 0,Y 523.368,Z 479.66,A -85,B 0,C 180,E1 -4773.079,E2 -4773.079} C_VEL
LIN {X 0,Y 523.427,Z 476.718,A -85,B 0,C 180,E1 -4774.235,E2 -4774.235} C_VEL
LIN {X 0,Y 523.463,Z 472.735,A -85,B 0,C 180,E1 -4775.393,E2 -4775.393} C_VEL
LIN {X 0,Y 523.516,Z 467.501,A -85,B 0,C 180,E1 -4776.574,E2 -4776.574} C_VEL
LIN {X 0,Y 523.625,Z 462.348,A -85,B 0,C 180,E1 -4777.519,E2 -4777.519} C_VEL
LIN {X 0,Y 523.784,Z 456.031,A -85,B 0,C 180,E1 -4778.488,E2 -4778.488} C_VEL
LIN {X 0,Y 523.921,Z 450.079,A -85,B 0,C 180,E1 -4779.263,E2 -4779.263} C_VEL
LIN {X 0,Y 524.084,Z 443.15,A -85,B 0,C 180,E1 -4780.04,E2 -4780.04} C_VEL
LIN {X 0,Y 524.345,Z 434.968,A -85,B 0,C 180,E1 -4780.815,E2 -4780.815} C_VEL
LIN {X 0,Y 524.534,Z 426.452,A -85,B 0,C 180,E1 -4781.496,E2 -4781.496} C_VEL
LIN {X 0,Y 524.713,Z 417.322,A -85,B 0,C 180,E1 -4782.105,E2 -4782.105} C_VEL
LIN {X 0,Y 524.953,Z 407.968,A -85,B 0,C 180,E1 -4782.614,E2 -4782.614} C_VEL
LIN {X 0,Y 525.133,Z 399.17,A -85,B 0,C 180,E1 -4783.003,E2 -4783.003} C_VEL
LIN {X 0,Y 525.314,Z 388.8,A -85,B 0,C 180,E1 -4783.355,E2 -4783.355} C_VEL
LIN {X 0,Y 523.546,Z 378.494,A -85,B 0,C 180,E1 -4783.652,E2 -4783.652} C_VEL
LIN {X 0,Y 523.411,Z 377.179,A -85,B 0,C 180,E1 -4783.689,E2 -4783.689} C_VEL
LIN {X 0,Y 523.421,Z 371.102,A -85,B 0,C 180,E1 -4786.378,E2 -4786.378} C_VEL
LIN {X 0,Y 523.515,Z 365.676,A -85,B 0,C 180,E1 -4788.795,E2 -4788.795} C_VEL
LIN {X 0,Y 523.573,Z 360.299,A -85,B 0,C 180,E1 -4791.249,E2 -4791.249} C_VEL
LIN {X 0,Y 523.667,Z 354.19,A -85,B 0,C 180,E1 -4794.131,E2 -4794.131} C_VEL
LIN {X 0,Y 523.776,Z 349.768,A -85,B 0,C 180,E1 -4796.282,E2 -4796.282} C_VEL
LIN {X 0,Y 523.948,Z 343.762,A -85,B 0,C 180,E1 -4799.322,E2 -4799.322} C_VEL
LIN {X 0,Y 524.089,Z 338.047,A -85,B 0,C 180,E1 -4802.346,E2 -4802.346} C_VEL
LIN {X 0,Y 524.262,Z 332.972,A -85,B 0,C 180,E1 -4805.2,E2 -4805.2} C_VEL
LIN {X 0,Y 524.365,Z 328.148,A -85,B 0,C 180,E1 -4808.063,E2 -4808.063} C_VEL
LIN {X 0,Y 524.521,Z 323.489,A -85,B 0,C 180,E1 -4811.037,E2 -4811.037} C_VEL
LIN {X 0,Y 524.433,Z 320.443,A -85,B 0,C 180,E1 -4813.114,E2 -4813.114} C_VEL
LIN {X 0,Y 523.962,Z 316.899,A -85,B 0,C 180,E1 -4815.774,E2 -4815.774} C_VEL
LIN {X 0,Y 523.94,Z 316.72,A -85,B 0,C 180,E1 -4818.907,E2 -4818.907} C_VEL
LIN {X 0,Y 523.917,Z 316.726,A -85,B 0,C 180,E1 -4821.898,E2 -4821.898} C_VEL
LIN {X 0,Y 523.925,Z 316.72,A -85,B 0,C 180,E1 -4824.911,E2 -4824.911} C_VEL
LIN {X 0,Y 523.936,Z 316.721,A -85,B 0,C 180,E1 -4827.679,E2 -4827.679} C_VEL
LIN {X 0,Y 523.954,Z 316.714,A -85,B 0,C 180,E1 -4830.676,E2 -4830.676} C_VEL
LIN {X 0,Y 523.974,Z 316.719,A -85,B 0,C 180,E1 -4833.728,E2 -4833.728} C_VEL
LIN {X 0,Y 523.913,Z 316.721,A -85,B 0,C 180,E1 -4836.269,E2 -4836.269} C_VEL
LIN {X 0,Y 523.945,Z 316.715,A -85,B 0,C 180,E1 -4838.766,E2 -4838.766} C_VEL
LIN {X 0,Y 523.948,Z 316.718,A -85,B 0,C 180,E1 -4841.22,E2 -4841.22} C_VEL
LIN {X 0,Y 523.933,Z 316.725,A -85,B 0,C 180,E1 -4843.638,E2 -4843.638} C_VEL
LIN {X 0,Y 523.944,Z 316.717,A -85,B 0,C 180,E1 -4846.028,E2 -4846.028} C_VEL
LIN {X 0,Y 524.012,Z 316.707,A -85,B 0,C 180,E1 -4848.394,E2 -4848.394} C_VEL
LIN {X 0,Y 524.004,Z 316.715,A -85,B 0,C 180,E1 -4851.516,E2 -4851.516} C_VEL
LIN {X 0,Y 524.082,Z 316.699,A -85,B 0,C 180,E1 -4854.613,E2 -4854.613} C_VEL
LIN {X 0,Y 524.113,Z 316.697,A -85,B 0,C 180,E1 -4857.694,E2 -4857.694} C_VEL
LIN {X 0,Y 524.121,Z 316.697,A -85,B 0,C 180,E1 -4860.768,E2 -4860.768} C_VEL
LIN {X 0,Y 524.071,Z 316.708,A -85,B 0,C 180,E1 -4863.074,E2 -4863.074} C_VEL
LIN {X 0,Y 524.037,Z 316.704,A -85,B 0,C 180,E1 -4866.159,E2 -4866.159} C_VEL
LIN {X 0,Y 524.002,Z 316.71,A -85,B 0,C 180,E1 -4868.484,E2 -4868.484} C_VEL
LIN {X 0,Y 524.001,Z 316.708,A -85,B 0,C 180,E1 -4871.739,E2 -4871.739} C_VEL
LIN {X 0,Y 523.991,Z 316.715,A -85,B 0,C 180,E1 -4875.052,E2 -4875.052} C_VEL
LIN {X 0,Y 523.962,Z 316.713,A -85,B 0,C 180,E1 -4877.969,E2 -4877.969} C_VEL
LIN {X 0,Y 523.97,Z 316.717,A -85,B 0,C 180,E1 -4880.41,E2 -4880.41} C_VEL
LIN {X 0,Y 523.909,Z 316.725,A -85,B 0,C 180,E1 -4882.893,E2 -4882.893} C_VEL
LIN {X 0,Y 523.95,Z 316.715,A -85,B 0,C 180,E1 -4885.418,E2 -4885.418} C_VEL
LIN {X 0,Y 523.967,Z 316.715,A -85,B 0,C 180,E1 -4887.999,E2 -4887.999} C_VEL
LIN {X 0,Y 523.944,Z 316.718,A -85,B 0,C 180,E1 -4890.855,E2 -4890.855} C_VEL
LIN {X 0,Y 523.957,Z 316.715,A -85,B 0,C 180,E1 -4893.734,E2 -4893.734} C_VEL
LIN {X 0,Y 523.917,Z 316.726,A -85,B 0,C 180,E1 -4896.404,E2 -4896.404} C_VEL
LIN {X 0,Y 523.929,Z 316.717,A -85,B 0,C 180,E1 -4899.083,E2 -4899.083} C_VEL
LIN {X 0,Y 523.954,Z 316.723,A -85,B 0,C 180,E1 -4902.118,E2 -4902.118} C_VEL
LIN {X 0,Y 523.952,Z 316.715,A -85,B 0,C 180,E1 -4905.308,E2 -4905.308} C_VEL
LIN {X 0,Y 523.916,Z 316.719,A -85,B 0,C 180,E1 -4906.899,E2 -4906.899} C_VEL
LIN {X 0,Y 523.254,Z 316.805,A -85,B 0,C 180,E1 -4907.541,E2 -4907.541} C_VEL
LIN {X 0,Y 520.427,Z 317.161,A -85,B 0,C 180,E1 -4908.583,E2 -4908.583} C_VEL
LIN {X 0,Y 518.03,Z 317.462,A -85,B 0,C 180,E1 -4909.422,E2 -4909.422} C_VEL
LIN {X 0,Y 516.99,Z 317.589,A -85,B 0,C 180,E1 -4910.07,E2 -4910.07} C_VEL
LIN {X 0,Y 516.899,Z 317.597,A -85,B 0,C 180,E1 -4910.289,E2 -4910.289} C_VEL
LIN {X 0,Y 516.88,Z 317.597,A -85,B 0,C 180,E1 -4913.342,E2 -4913.342} C_VEL
LIN {X 0,Y 516.907,Z 317.596,A -85,B 0,C 180,E1 -4916.121,E2 -4916.121} C_VEL
LIN {X 0,Y 516.889,Z 317.594,A -85,B 0,C 180,E1 -4918.935,E2 -4918.935} C_VEL
LIN {X 0,Y 516.917,Z 317.598,A -85,B 0,C 180,E1 -4921.585,E2 -4921.585} C_VEL
LIN {X 0,Y 516.93,Z 317.59,A -85,B 0,C 180,E1 -4924.211,E2 -4924.211} C_VEL
LIN {X 0,Y 516.862,Z 317.598,A -85,B 0,C 180,E1 -4926.776,E2 -4926.776} C_VEL
LIN {X 0,Y 516.936,Z 317.594,A -85,B 0,C 180,E1 -4929.731,E2 -4929.731} C_VEL
LIN {X 0,Y 516.926,Z 317.592,A -85,B 0,C 180,E1 -4932.596,E2 -4932.596} C_VEL
LIN {X 0,Y 516.948,Z 317.593,A -85,B 0,C 180,E1 -4935.03,E2 -4935.03} C_VEL
LIN {X 0,Y 516.962,Z 317.586,A -85,B 0,C 180,E1 -4938.234,E2 -4938.234} C_VEL
LIN {X 0,Y 516.967,Z 317.592,A -85,B 0,C 180,E1 -4941.4,E2 -4941.4} C_VEL
LIN {X 0,Y 517.013,Z 317.582,A -85,B 0,C 180,E1 -4943.757,E2 -4943.757} C_VEL
LIN {X 0,Y 517.083,Z 317.573,A -85,B 0,C 180,E1 -4947.663,E2 -4947.663} C_VEL
LIN {X 0,Y 517.091,Z 317.576,A -85,B 0,C 180,E1 -4950.779,E2 -4950.779} C_VEL
LIN {X 0,Y 517.01,Z 317.587,A -85,B 0,C 180,E1 -4953.117,E2 -4953.117} C_VEL
LIN {X 0,Y 517.013,Z 317.582,A -85,B 0,C 180,E1 -4956.243,E2 -4956.243} C_VEL
LIN {X 0,Y 516.951,Z 317.59,A -85,B 0,C 180,E1 -4959.389,E2 -4959.389} C_VEL
LIN {X 0,Y 516.949,Z 317.588,A -85,B 0,C 180,E1 -4961.808,E2 -4961.808} C_VEL
LIN {X 0,Y 516.944,Z 317.591,A -85,B 0,C 180,E1 -4965.148,E2 -4965.148} C_VEL
LIN {X 0,Y 516.922,Z 317.596,A -85,B 0,C 180,E1 -4968.222,E2 -4968.222} C_VEL
LIN {X 0,Y 516.909,Z 317.597,A -85,B 0,C 180,E1 -4970.702,E2 -4970.702} C_VEL
LIN {X 0,Y 516.9,Z 317.597,A -85,B 0,C 180,E1 -4974.072,E2 -4974.072} C_VEL
LIN {X 0,Y 516.926,Z 317.594,A -85,B 0,C 180,E1 -4976.658,E2 -4976.658} C_VEL
LIN {X 0,Y 516.908,Z 317.592,A -85,B 0,C 180,E1 -4979.524,E2 -4979.524} C_VEL
LIN {X 0,Y 516.897,Z 317.597,A -85,B 0,C 180,E1 -4982.544,E2 -4982.544} C_VEL
LIN {X 0,Y 516.875,Z 317.596,A -85,B 0,C 180,E1 -4985.332,E2 -4985.332} C_VEL
LIN {X 0,Y 516.878,Z 317.602,A -85,B 0,C 180,E1 -4987.944,E2 -4987.944} C_VEL
LIN {X 0,Y 516.901,Z 317.593,A -85,B 0,C 180,E1 -4990.74,E2 -4990.74} C_VEL
LIN {X 0,Y 516.879,Z 317.604,A -85,B 0,C 180,E1 -4993.903,E2 -4993.903} C_VEL
LIN {X 0,Y 516.879,Z 317.601,A -85,B 0,C 180,E1 -4996.107,E2 -4996.107} C_VEL
LIN {X 0,Y 516.901,Z 317.594,A -85,B 0,C 180,E1 -4999.261,E2 -4999.261} C_VEL
LIN {X 0,Y 516.861,Z 317.599,A -85,B 0,C 180,E1 -5002.275,E2 -5002.275} C_VEL
LIN {X 0,Y 516.88,Z 317.598,A -85,B 0,C 180,E1 -5005.176,E2 -5005.176} C_VEL
LIN {X 0,Y 516.88,Z 317.599,A -85,B 0,C 180,E1 -5007.976,E2 -5007.976} C_VEL
LIN {X 0,Y 516.919,Z 317.591,A -85,B 0,C 180,E1 -5010.696,E2 -5010.696} C_VEL
LIN {X 0,Y 516.94,Z 317.592,A -85,B 0,C 180,E1 -5013.804,E2 -5013.804} C_VEL
LIN {X 0,Y 516.863,Z 317.599,A -85,B 0,C 180,E1 -5016.777,E2 -5016.777} C_VEL
LIN {X 0,Y 516.937,Z 317.591,A -85,B 0,C 180,E1 -5019.732,E2 -5019.732} C_VEL
LIN {X 0,Y 516.927,Z 317.59,A -85,B 0,C 180,E1 -5022.597,E2 -5022.597} C_VEL
LIN {X 0,Y 516.94,Z 317.594,A -85,B 0,C 180,E1 -5025.031,E2 -5025.031} C_VEL
LIN {X 0,Y 516.964,Z 317.585,A -85,B 0,C 180,E1 -5028.234,E2 -5028.234} C_VEL
LIN {X 0,Y 516.967,Z 317.588,A -85,B 0,C 180,E1 -5031.4,E2 -5031.4} C_VEL
LIN {X 0,Y 517.002,Z 317.58,A -85,B 0,C 180,E1 -5033.757,E2 -5033.757} C_VEL
LIN {X 0,Y 517.012,Z 317.588,A -85,B 0,C 180,E1 -5036.883,E2 -5036.883} C_VEL
LIN {X 0,Y 517.085,Z 317.57,A -85,B 0,C 180,E1 -5040,E2 -5040} C_VEL
LIN {X 0,Y 517.01,Z 317.583,A -85,B 0,C 180,E1 -5043.117,E2 -5043.117} C_VEL
LIN {X 0,Y 517.003,Z 317.583,A -85,B 0,C 180,E1 -5046.244,E2 -5046.244} C_VEL
LIN {X 0,Y 516.953,Z 317.586,A -85,B 0,C 180,E1 -5049.39,E2 -5049.39} C_VEL
LIN {X 0,Y 516.952,Z 317.587,A -85,B 0,C 180,E1 -5051.808,E2 -5051.808} C_VEL
LIN {X 0,Y 516.947,Z 317.588,A -85,B 0,C 180,E1 -5055.148,E2 -5055.148} C_VEL
LIN {X 0,Y 516.916,Z 317.597,A -85,B 0,C 180,E1 -5058.223,E2 -5058.223} C_VEL
LIN {X 0,Y 516.912,Z 317.595,A -85,B 0,C 180,E1 -5060.702,E2 -5060.702} C_VEL
LIN {X 0,Y 516.891,Z 317.6,A -85,B 0,C 180,E1 -5064.073,E2 -5064.073} C_VEL
LIN {X 0,Y 516.925,Z 317.592,A -85,B 0,C 180,E1 -5066.658,E2 -5066.658} C_VEL
LIN {X 0,Y 516.911,Z 317.593,A -85,B 0,C 180,E1 -5069.524,E2 -5069.524} C_VEL
LIN {X 0,Y 516.896,Z 317.595,A -85,B 0,C 180,E1 -5072.544,E2 -5072.544} C_VEL
LIN {X 0,Y 516.867,Z 317.598,A -85,B 0,C 180,E1 -5075.33,E2 -5075.33} C_VEL
LIN {X 0,Y 516.882,Z 317.604,A -85,B 0,C 180,E1 -5077.944,E2 -5077.944} C_VEL
LIN {X 0,Y 516.884,Z 317.599,A -85,B 0,C 180,E1 -5080.742,E2 -5080.742} C_VEL
LIN {X 0,Y 516.883,Z 317.601,A -85,B 0,C 180,E1 -5082.832,E2 -5082.832} C_VEL
LIN {X 0,Y 516.893,Z 317.726,A -85,B 0,C 180,E1 -5083.903,E2 -5083.903} C_VEL
LIN {X 0,Y 517.318,Z 320.647,A -85,B 0,C 180,E1 -5086.144,E2 -5086.144} C_VEL
LIN {X 0,Y 517.513,Z 323.7,A -85,B 0,C 180,E1 -5088.325,E2 -5088.325} C_VEL
LIN {X 0,Y 517.427,Z 328.293,A -85,B 0,C 180,E1 -5091.333,E2 -5091.333} C_VEL
LIN {X 0,Y 517.246,Z 333.06,A -85,B 0,C 180,E1 -5094.25,E2 -5094.25} C_VEL
LIN {X 0,Y 517.082,Z 337.959,A -85,B 0,C 180,E1 -5097.067,E2 -5097.067} C_VEL
LIN {X 0,Y 516.929,Z 342.977,A -85,B 0,C 180,E1 -5099.799,E2 -5099.799} C_VEL
LIN {X 0,Y 516.789,Z 348.051,A -85,B 0,C 180,E1 -5102.459,E2 -5102.459} C_VEL
LIN {X 0,Y 516.636,Z 353.223,A -85,B 0,C 180,E1 -5105.058,E2 -5105.058} C_VEL
LIN {X 0,Y 516.564,Z 358.647,A -85,B 0,C 180,E1 -5107.693,E2 -5107.693} C_VEL
LIN {X 0,Y 516.488,Z 363.766,A -85,B 0,C 180,E1 -5110.112,E2 -5110.112} C_VEL
LIN {X 0,Y 516.419,Z 369.111,A -85,B 0,C 180,E1 -5112.579,E2 -5112.579} C_VEL
LIN {X 0,Y 516.321,Z 376.319,A -85,B 0,C 180,E1 -5115.818,E2 -5115.818} C_VEL
LIN {X 0,Y 516.333,Z 377.122,A -85,B 0,C 180,E1 -5116.132,E2 -5116.132} C_VEL
LIN {X 0,Y 517.91,Z 386.732,A -85,B 0,C 180,E1 -5116.397,E2 -5116.397} C_VEL
LIN {X 0,Y 518.396,Z 390.791,A -85,B 0,C 180,E1 -5116.525,E2 -5116.525} C_VEL
LIN {X 0,Y 518.097,Z 403.741,A -85,B 0,C 180,E1 -5117.017,E2 -5117.017} C_VEL
LIN {X 0,Y 517.846,Z 415.106,A -85,B 0,C 180,E1 -5117.609,E2 -5117.609} C_VEL
LIN {X 0,Y 517.59,Z 423.212,A -85,B 0,C 180,E1 -5118.124,E2 -5118.124} C_VEL
LIN {X 0,Y 517.383,Z 432.5,A -85,B 0,C 180,E1 -5118.839,E2 -5118.839} C_VEL
LIN {X 0,Y 517.143,Z 441.034,A -85,B 0,C 180,E1 -5119.626,E2 -5119.626} C_VEL
LIN {X 0,Y 516.956,Z 448.256,A -85,B 0,C 180,E1 -5120.413,E2 -5120.413} C_VEL
LIN {X 0,Y 516.739,Z 454.458,A -85,B 0,C 180,E1 -5121.199,E2 -5121.199} C_VEL
LIN {X 0,Y 516.595,Z 460.996,A -85,B 0,C 180,E1 -5122.181,E2 -5122.181} C_VEL
LIN {X 0,Y 516.481,Z 466.644,A -85,B 0,C 180,E1 -5123.201,E2 -5123.201} C_VEL
LIN {X 0,Y 516.429,Z 470.987,A -85,B 0,C 180,E1 -5124.142,E2 -5124.142} C_VEL
LIN {X 0,Y 516.277,Z 475.305,A -85,B 0,C 180,E1 -5125.315,E2 -5125.315} C_VEL
LIN {X 0,Y 516.353,Z 477.671,A -85,B 0,C 180,E1 -5126.098,E2 -5126.098} C_VEL
LIN {X 0,Y 516.283,Z 479.465,A -85,B 0,C 180,E1 -5126.879,E2 -5126.879} C_VEL
LIN {X 0,Y 516.192,Z 481.902,A -85,B 0,C 180,E1 -5128.44,E2 -5128.44} C_VEL
LIN {X 0,Y 516.16,Z 482.488,A -85,B 0,C 180,E1 -5129.22,E2 -5129.22} C_VEL
LIN {X 0,Y 516.16,Z 482.488,A -85,B 0,C 180,E1 -5130.78,E2 -5130.78} C_VEL
LIN {X 0,Y 516.192,Z 481.902,A -85,B 0,C 180,E1 -5131.56,E2 -5131.56} C_VEL
LIN {X 0,Y 516.283,Z 479.465,A -85,B 0,C 180,E1 -5133.121,E2 -5133.121} C_VEL
LIN {X 0,Y 516.316,Z 476.521,A -85,B 0,C 180,E1 -5134.293,E2 -5134.293} C_VEL
LIN {X 0,Y 516.379,Z 472.538,A -85,B 0,C 180,E1 -5135.467,E2 -5135.467} C_VEL
LIN {X 0,Y 516.433,Z 467.788,A -85,B 0,C 180,E1 -5136.565,E2 -5136.565} C_VEL
LIN {X 0,Y 516.557,Z 462.151,A -85,B 0,C 180,E1 -5137.623,E2 -5137.623} C_VEL
LIN {X 0,Y 516.731,Z 455.835,A -85,B 0,C 180,E1 -5138.604,E2 -5138.604} C_VEL
LIN {X 0,Y 516.899,Z 449.883,A -85,B 0,C 180,E1 -5139.39,E2 -5139.39} C_VEL
LIN {X 0,Y 517.052,Z 442.952,A -85,B 0,C 180,E1 -5140.178,E2 -5140.178} C_VEL
LIN {X 0,Y 517.338,Z 434.771,A -85,B 0,C 180,E1 -5140.964,E2 -5140.964} C_VEL
LIN {X 0,Y 517.551,Z 426.256,A -85,B 0,C 180,E1 -5141.653,E2 -5141.653} C_VEL
LIN {X 0,Y 517.719,Z 418.211,A -85,B 0,C 180,E1 -5142.205,E2 -5142.205} C_VEL
LIN {X 0,Y 517.99,Z 408.779,A -85,B 0,C 180,E1 -5142.737,E2 -5142.737} C_VEL
LIN {X 0,Y 518.208,Z 398.974,A -85,B 0,C 180,E1 -5143.18,E2 -5143.18} C_VEL
LIN {X 0,Y 518.345,Z 389.478,A -85,B 0,C 180,E1 -5143.513,E2 -5143.513} C_VEL
LIN {X 0,Y 516.467,Z 378.428,A -85,B 0,C 180,E1 -5143.84,E2 -5143.84} C_VEL
LIN {X 0,Y 516.311,Z 376.993,A -85,B 0,C 180,E1 -5143.881,E2 -5143.881} C_VEL
LIN {X 0,Y 516.338,Z 370.913,A -85,B 0,C 180,E1 -5146.609,E2 -5146.609} C_VEL
LIN {X 0,Y 516.431,Z 365.539,A -85,B 0,C 180,E1 -5149.063,E2 -5149.063} C_VEL
LIN {X 0,Y 516.508,Z 360.219,A -85,B 0,C 180,E1 -5151.554,E2 -5151.554} C_VEL
LIN {X 0,Y 516.619,Z 354.532,A -85,B 0,C 180,E1 -5154.292,E2 -5154.292} C_VEL
LIN {X 0,Y 516.719,Z 349.759,A -85,B 0,C 180,E1 -5156.669,E2 -5156.669} C_VEL
LIN {X 0,Y 516.904,Z 344.221,A -85,B 0,C 180,E1 -5159.522,E2 -5159.522} C_VEL
LIN {X 0,Y 517.056,Z 338.584,A -85,B 0,C 180,E1 -5162.57,E2 -5162.57} C_VEL
LIN {X 0,Y 517.231,Z 333.658,A -85,B 0,C 180,E1 -5165.386,E2 -5165.386} C_VEL
LIN {X 0,Y 517.346,Z 329.309,A -85,B 0,C 180,E1 -5168.009,E2 -5168.009} C_VEL
LIN {X 0,Y 517.497,Z 325.16,A -85,B 0,C 180,E1 -5170.683,E2 -5170.683} C_VEL
LIN {X 0,Y 517.484,Z 322.033,A -85,B 0,C 180,E1 -5172.829,E2 -5172.829} C_VEL
LIN {X 0,Y 517.078,Z 319.09,A -85,B 0,C 180,E1 -5175.027,E2 -5175.027} C_VEL
LIN {X 0,Y 516.891,Z 317.71,A -85,B 0,C 180,E1 -5176.106,E2 -5176.106} C_VEL
LIN {X 0,Y 516.914,Z 317.598,A -85,B 0,C 180,E1 -5178.398,E2 -5178.398} C_VEL
LIN {X 0,Y 516.882,Z 317.598,A -85,B 0,C 180,E1 -5181.284,E2 -5181.284} C_VEL
LIN {X 0,Y 516.872,Z 317.605,A -85,B 0,C 180,E1 -5184.219,E2 -5184.219} C_VEL
LIN {X 0,Y 516.895,Z 317.593,A -85,B 0,C 180,E1 -5187.053,E2 -5187.053} C_VEL
LIN {X 0,Y 516.892,Z 317.601,A -85,B 0,C 180,E1 -5189.796,E2 -5189.796} C_VEL
LIN {X 0,Y 516.926,Z 317.591,A -85,B 0,C 180,E1 -5192.467,E2 -5192.467} C_VEL
LIN {X 0,Y 516.875,Z 317.596,A -85,B 0,C 180,E1 -5195.07,E2 -5195.07} C_VEL
LIN {X 0,Y 516.869,Z 317.604,A -85,B 0,C 180,E1 -5197.621,E2 -5197.621} C_VEL
LIN {X 0,Y 516.931,Z 317.591,A -85,B 0,C 180,E1 -5200.129,E2 -5200.129} C_VEL
LIN {X 0,Y 516.907,Z 317.592,A -85,B 0,C 180,E1 -5202.595,E2 -5202.595} C_VEL
LIN {X 0,Y 516.951,Z 317.588,A -85,B 0,C 180,E1 -5205.03,E2 -5205.03} C_VEL
LIN {X 0,Y 516.966,Z 317.585,A -85,B 0,C 180,E1 -5208.233,E2 -5208.233} C_VEL
LIN {X 0,Y 516.969,Z 317.593,A -85,B 0,C 180,E1 -5211.399,E2 -5211.399} C_VEL
LIN {X 0,Y 517.002,Z 317.583,A -85,B 0,C 180,E1 -5213.756,E2 -5213.756} C_VEL
LIN {X 0,Y 517.01,Z 317.583,A -85,B 0,C 180,E1 -5216.883,E2 -5216.883} C_VEL
LIN {X 0,Y 517.085,Z 317.57,A -85,B 0,C 180,E1 -5220,E2 -5220} C_VEL
LIN {X 0,Y 517.012,Z 317.588,A -85,B 0,C 180,E1 -5223.117,E2 -5223.117} C_VEL
LIN {X 0,Y 517.002,Z 317.58,A -85,B 0,C 180,E1 -5226.243,E2 -5226.243} C_VEL
LIN {X 0,Y 516.95,Z 317.589,A -85,B 0,C 180,E1 -5229.389,E2 -5229.389} C_VEL
LIN {X 0,Y 516.95,Z 317.586,A -85,B 0,C 180,E1 -5231.807,E2 -5231.807} C_VEL
LIN {X 0,Y 516.943,Z 317.591,A -85,B 0,C 180,E1 -5235.146,E2 -5235.146} C_VEL
LIN {X 0,Y 516.923,Z 317.592,A -85,B 0,C 180,E1 -5238.222,E2 -5238.222} C_VEL
LIN {X 0,Y 516.91,Z 317.6,A -85,B 0,C 180,E1 -5240.701,E2 -5240.701} C_VEL
LIN {X 0,Y 516.901,Z 317.595,A -85,B 0,C 180,E1 -5244.072,E2 -5244.072} C_VEL
LIN {X 0,Y 516.923,Z 317.597,A -85,B 0,C 180,E1 -5246.657,E2 -5246.657} C_VEL
LIN {X 0,Y 516.908,Z 317.592,A -85,B 0,C 180,E1 -5249.523,E2 -5249.523} C_VEL
LIN {X 0,Y 516.898,Z 317.6,A -85,B 0,C 180,E1 -5252.544,E2 -5252.544} C_VEL
LIN {X 0,Y 516.876,Z 317.596,A -85,B 0,C 180,E1 -5255.331,E2 -5255.331} C_VEL
LIN {X 0,Y 516.879,Z 317.6,A -85,B 0,C 180,E1 -5257.943,E2 -5257.943} C_VEL
LIN {X 0,Y 516.901,Z 317.594,A -85,B 0,C 180,E1 -5260.739,E2 -5260.739} C_VEL
LIN {X 0,Y 516.879,Z 317.601,A -85,B 0,C 180,E1 -5263.903,E2 -5263.903} C_VEL
LIN {X 0,Y 516.878,Z 317.604,A -85,B 0,C 180,E1 -5266.107,E2 -5266.107} C_VEL
LIN {X 0,Y 516.901,Z 317.593,A -85,B 0,C 180,E1 -5269.26,E2 -5269.26} C_VEL
LIN {X 0,Y 516.899,Z 317.597,A -85,B 0,C 180,E1 -5270.289,E2 -5270.289} C_VEL
LIN {X 0,Y 516.218,Z 317.679,A -85,B 0,C 180,E1 -5270.939,E2 -5270.939} C_VEL
LIN {X 0,Y 513.365,Z 318.041,A -85,B 0,C 180,E1 -5271.994,E2 -5271.994} C_VEL
LIN {X 0,Y 510.957,Z 318.343,A -85,B 0,C 180,E1 -5272.844,E2 -5272.844} C_VEL
LIN {X 0,Y 509.916,Z 318.469,A -85,B 0,C 180,E1 -5273.5,E2 -5273.5} C_VEL
LIN {X 0,Y 509.827,Z 318.478,A -85,B 0,C 180,E1 -5273.723,E2 -5273.723} C_VEL
LIN {X 0,Y 509.858,Z 318.471,A -85,B 0,C 180,E1 -5276.539,E2 -5276.539} C_VEL
LIN {X 0,Y 509.843,Z 318.475,A -85,B 0,C 180,E1 -5279.334,E2 -5279.334} C_VEL
LIN {X 0,Y 509.892,Z 318.469,A -85,B 0,C 180,E1 -5282.055,E2 -5282.055} C_VEL
LIN {X 0,Y 509.874,Z 318.468,A -85,B 0,C 180,E1 -5284.704,E2 -5284.704} C_VEL
LIN {X 0,Y 509.823,Z 318.482,A -85,B 0,C 180,E1 -5287.458,E2 -5287.458} C_VEL
LIN {X 0,Y 509.913,Z 318.467,A -85,B 0,C 180,E1 -5289.845,E2 -5289.845} C_VEL
LIN {X 0,Y 509.881,Z 318.474,A -85,B 0,C 180,E1 -5293.175,E2 -5293.175} C_VEL
LIN {X 0,Y 509.87,Z 318.475,A -85,B 0,C 180,E1 -5295.634,E2 -5295.634} C_VEL
LIN {X 0,Y 509.911,Z 318.468,A -85,B 0,C 180,E1 -5298.875,E2 -5298.875} C_VEL
LIN {X 0,Y 509.949,Z 318.461,A -85,B 0,C 180,E1 -5302.078,E2 -5302.078} C_VEL
LIN {X 0,Y 509.983,Z 318.458,A -85,B 0,C 180,E1 -5304.464,E2 -5304.464} C_VEL
LIN {X 0,Y 510.054,Z 318.449,A -85,B 0,C 180,E1 -5307.631,E2 -5307.631} C_VEL
LIN {X 0,Y 510.061,Z 318.452,A -85,B 0,C 180,E1 -5310.789,E2 -5310.789} C_VEL
LIN {X 0,Y 509.953,Z 318.466,A -85,B 0,C 180,E1 -5313.16,E2 -5313.16} C_VEL
LIN {X 0,Y 509.98,Z 318.459,A -85,B 0,C 180,E1 -5316.33,E2 -5316.33} C_VEL
LIN {X 0,Y 509.913,Z 318.472,A -85,B 0,C 180,E1 -5318.72,E2 -5318.72} C_VEL
LIN {X 0,Y 509.901,Z 318.466,A -85,B 0,C 180,E1 -5321.932,E2 -5321.932} C_VEL
LIN {X 0,Y 509.89,Z 318.469,A -85,B 0,C 180,E1 -5325.242,E2 -5325.242} C_VEL
LIN {X 0,Y 509.885,Z 318.47,A -85,B 0,C 180,E1 -5328.001,E2 -5328.001} C_VEL
LIN {X 0,Y 509.847,Z 318.473,A -85,B 0,C 180,E1 -5331.002,E2 -5331.002} C_VEL
LIN {X 0,Y 509.862,Z 318.478,A -85,B 0,C 180,E1 -5334.426,E2 -5334.426} C_VEL
LIN {X 0,Y 509.884,Z 318.467,A -85,B 0,C 180,E1 -5337.056,E2 -5337.056} C_VEL
LIN {X 0,Y 509.854,Z 318.472,A -85,B 0,C 180,E1 -5339.751,E2 -5339.751} C_VEL
LIN {X 0,Y 509.873,Z 318.47,A -85,B 0,C 180,E1 -5342.775,E2 -5342.775} C_VEL
LIN {X 0,Y 509.836,Z 318.474,A -85,B 0,C 180,E1 -5345.581,E2 -5345.581} C_VEL
LIN {X 0,Y 509.849,Z 318.476,A -85,B 0,C 180,E1 -5348.338,E2 -5348.338} C_VEL
LIN {X 0,Y 509.862,Z 318.471,A -85,B 0,C 180,E1 -5351.425,E2 -5351.425} C_VEL
LIN {X 0,Y 509.853,Z 318.471,A -85,B 0,C 180,E1 -5354.668,E2 -5354.668} C_VEL
LIN {X 0,Y 509.878,Z 318.472,A -85,B 0,C 180,E1 -5358.1,E2 -5358.1} C_VEL
LIN {X 0,Y 509.857,Z 318.47,A -85,B 0,C 180,E1 -5360.649,E2 -5360.649} C_VEL
LIN {X 0,Y 509.821,Z 318.483,A -85,B 0,C 180,E1 -5363.647,E2 -5363.647} C_VEL
LIN {X 0,Y 509.857,Z 318.47,A -85,B 0,C 180,E1 -5366.54,E2 -5366.54} C_VEL
LIN {X 0,Y 509.843,Z 318.477,A -85,B 0,C 180,E1 -5369.335,E2 -5369.335} C_VEL
LIN {X 0,Y 509.891,Z 318.468,A -85,B 0,C 180,E1 -5372.055,E2 -5372.055} C_VEL
LIN {X 0,Y 509.873,Z 318.469,A -85,B 0,C 180,E1 -5374.704,E2 -5374.704} C_VEL
LIN {X 0,Y 509.824,Z 318.482,A -85,B 0,C 180,E1 -5377.458,E2 -5377.458} C_VEL
LIN {X 0,Y 509.915,Z 318.465,A -85,B 0,C 180,E1 -5379.845,E2 -5379.845} C_VEL
LIN {X 0,Y 509.882,Z 318.475,A -85,B 0,C 180,E1 -5383.175,E2 -5383.175} C_VEL
LIN {X 0,Y 509.862,Z 318.472,A -85,B 0,C 180,E1 -5385.635,E2 -5385.635} C_VEL
LIN {X 0,Y 509.912,Z 318.469,A -85,B 0,C 180,E1 -5388.875,E2 -5388.875} C_VEL
LIN {X 0,Y 509.95,Z 318.458,A -85,B 0,C 180,E1 -5392.079,E2 -5392.079} C_VEL
LIN {X 0,Y 509.979,Z 318.457,A -85,B 0,C 180,E1 -5394.465,E2 -5394.465} C_VEL
LIN {X 0,Y 510.055,Z 318.446,A -85,B 0,C 180,E1 -5397.631,E2 -5397.631} C_VEL
LIN {X 0,Y 510.063,Z 318.453,A -85,B 0,C 180,E1 -5400.79,E2 -5400.79} C_VEL
LIN {X 0,Y 509.953,Z 318.461,A -85,B 0,C 180,E1 -5403.161,E2 -5403.161} C_VEL
LIN {X 0,Y 509.954,Z 318.462,A -85,B 0,C 180,E1 -5406.33,E2 -5406.33} C_VEL
LIN {X 0,Y 509.915,Z 318.47,A -85,B 0,C 180,E1 -5408.721,E2 -5408.721} C_VEL
LIN {X 0,Y 509.904,Z 318.466,A -85,B 0,C 180,E1 -5411.932,E2 -5411.932} C_VEL
LIN {X 0,Y 509.894,Z 318.466,A -85,B 0,C 180,E1 -5415.242,E2 -5415.242} C_VEL
LIN {X 0,Y 509.867,Z 318.472,A -85,B 0,C 180,E1 -5417.994,E2 -5417.994} C_VEL
LIN {X 0,Y 509.886,Z 318.474,A -85,B 0,C 180,E1 -5420.402,E2 -5420.402} C_VEL
LIN {X 0,Y 509.822,Z 318.475,A -85,B 0,C 180,E1 -5423.564,E2 -5423.564} C_VEL
LIN {X 0,Y 509.911,Z 318.469,A -85,B 0,C 180,E1 -5426.379,E2 -5426.379} C_VEL
LIN {X 0,Y 509.877,Z 318.468,A -85,B 0,C 180,E1 -5428.845,E2 -5428.845} C_VEL
LIN {X 0,Y 509.821,Z 318.477,A -85,B 0,C 180,E1 -5431.591,E2 -5431.591} C_VEL
LIN {X 0,Y 509.848,Z 318.475,A -85,B 0,C 180,E1 -5434.414,E2 -5434.414} C_VEL
LIN {X 0,Y 509.818,Z 318.479,A -85,B 0,C 180,E1 -5437.341,E2 -5437.341} C_VEL
LIN {X 0,Y 509.839,Z 318.478,A -85,B 0,C 180,E1 -5440.383,E2 -5440.383} C_VEL
LIN {X 0,Y 509.823,Z 318.481,A -85,B 0,C 180,E1 -5443.062,E2 -5443.062} C_VEL
LIN {X 0,Y 509.824,Z 318.543,A -85,B 0,C 180,E1 -5443.572,E2 -5443.572} C_VEL
LIN {X 0,Y 510.358,Z 322.28,A -85,B 0,C 180,E1 -5446.486,E2 -5446.486} C_VEL
LIN {X 0,Y 510.484,Z 325.318,A -85,B 0,C 180,E1 -5448.637,E2 -5448.637} C_VEL
LIN {X 0,Y 510.391,Z 329.954,A -85,B 0,C 180,E1 -5451.71,E2 -5451.71} C_VEL
LIN {X 0,Y 510.2,Z 334.753,A -85,B 0,C 180,E1 -5454.652,E2 -5454.652} C_VEL
LIN {X 0,Y 510.019,Z 339.642,A -85,B 0,C 180,E1 -5457.492,E2 -5457.492} C_VEL
LIN {X 0,Y 509.864,Z 344.698,A -85,B 0,C 180,E1 -5460.273,E2 -5460.273} C_VEL
LIN {X 0,Y 509.693,Z 349.755,A -85,B 0,C 180,E1 -5462.933,E2 -5462.933} C_VEL
LIN {X 0,Y 509.556,Z 354.913,A -85,B 0,C 180,E1 -5465.558,E2 -5465.558} C_VEL
LIN {X 0,Y 509.445,Z 360.152,A -85,B 0,C 180,E1 -5468.132,E2 -5468.132} C_VEL
LIN {X 0,Y 509.356,Z 365.441,A -85,B 0,C 180,E1 -5470.662,E2 -5470.662} C_VEL
LIN {X 0,Y 509.286,Z 370.771,A -85,B 0,C 180,E1 -5473.154,E2 -5473.154} C_VEL
LIN {X 0,Y 509.248,Z 376.821,A -85,B 0,C 180,E1 -5475.922,E2 -5475.922} C_VEL
LIN {X 0,Y 511.163,Z 388.618,A -85,B 0,C 180,E1 -5476.274,E2 -5476.274} C_VEL
LIN {X 0,Y 511.437,Z 393.626,A -85,B 0,C 180,E1 -5476.44,E2 -5476.44} C_VEL
LIN {X 0,Y 511.158,Z 404.553,A -85,B 0,C 180,E1 -5476.888,E2 -5476.888} C_VEL
LIN {X 0,Y 510.887,Z 414.952,A -85,B 0,C 180,E1 -5477.44,E2 -5477.44} C_VEL
LIN {X 0,Y 510.606,Z 423.452,A -85,B 0,C 180,E1 -5477.992,E2 -5477.992} C_VEL
LIN {X 0,Y 510.397,Z 432.304,A -85,B 0,C 180,E1 -5478.684,E2 -5478.684} C_VEL
LIN {X 0,Y 510.106,Z 440.836,A -85,B 0,C 180,E1 -5479.482,E2 -5479.482} C_VEL
LIN {X 0,Y 509.904,Z 448.058,A -85,B 0,C 180,E1 -5480.28,E2 -5480.28} C_VEL
LIN {X 0,Y 509.691,Z 454.261,A -85,B 0,C 180,E1 -5481.076,E2 -5481.076} C_VEL
LIN {X 0,Y 509.535,Z 460.799,A -85,B 0,C 180,E1 -5482.072,E2 -5482.072} C_VEL
LIN {X 0,Y 509.403,Z 466.688,A -85,B 0,C 180,E1 -5483.156,E2 -5483.156} C_VEL
LIN {X 0,Y 509.339,Z 470.79,A -85,B 0,C 180,E1 -5484.06,E2 -5484.06} C_VEL
LIN {X 0,Y 509.193,Z 475.109,A -85,B 0,C 180,E1 -5485.25,E2 -5485.25} C_VEL
LIN {X 0,Y 509.247,Z 477.474,A -85,B 0,C 180,E1 -5486.043,E2 -5486.043} C_VEL
LIN {X 0,Y 509.201,Z 479.269,A -85,B 0,C 180,E1 -5486.835,E2 -5486.835} C_VEL
LIN {X 0,Y 509.113,Z 481.707,A -85,B 0,C 180,E1 -5488.418,E2 -5488.418} C_VEL
LIN {X 0,Y 509.074,Z 482.293,A -85,B 0,C 180,E1 -5489.209,E2 -5489.209} C_VEL
LIN {X 0,Y 509.074,Z 482.293,A -85,B 0,C 180,E1 -5490.791,E2 -5490.791} C_VEL
LIN {X 0,Y 509.113,Z 481.707,A -85,B 0,C 180,E1 -5491.582,E2 -5491.582} C_VEL
LIN {X 0,Y 509.201,Z 479.269,A -85,B 0,C 180,E1 -5493.165,E2 -5493.165} C_VEL
LIN {X 0,Y 509.208,Z 476.325,A -85,B 0,C 180,E1 -5494.353,E2 -5494.353} C_VEL
LIN {X 0,Y 509.297,Z 472.342,A -85,B 0,C 180,E1 -5495.543,E2 -5495.543} C_VEL
LIN {X 0,Y 509.35,Z 468.074,A -85,B 0,C 180,E1 -5496.557,E2 -5496.557} C_VEL
LIN {X 0,Y 509.469,Z 463.11,A -85,B 0,C 180,E1 -5497.53,E2 -5497.53} C_VEL
LIN {X 0,Y 509.644,Z 457.014,A -85,B 0,C 180,E1 -5498.525,E2 -5498.525} C_VEL
LIN {X 0,Y 509.789,Z 451.313,A -85,B 0,C 180,E1 -5499.322,E2 -5499.322} C_VEL
LIN {X 0,Y 510.032,Z 442.756,A -85,B 0,C 180,E1 -5500.319,E2 -5500.319} C_VEL
LIN {X 0,Y 510.34,Z 434.575,A -85,B 0,C 180,E1 -5501.116,E2 -5501.116} C_VEL
LIN {X 0,Y 510.581,Z 426.059,A -85,B 0,C 180,E1 -5501.815,E2 -5501.815} C_VEL
LIN {X 0,Y 510.778,Z 417.54,A -85,B 0,C 180,E1 -5502.402,E2 -5502.402} C_VEL
LIN {X 0,Y 511.048,Z 407.574,A -85,B 0,C 180,E1 -5502.964,E2 -5502.964} C_VEL
LIN {X 0,Y 511.313,Z 398.778,A -85,B 0,C 180,E1 -5503.361,E2 -5503.361} C_VEL
LIN {X 0,Y 511.387,Z 390.155,A -85,B 0,C 180,E1 -5503.675,E2 -5503.675} C_VEL
LIN {X 0,Y 509.534,Z 378.776,A -85,B 0,C 180,E1 -5504.022,E2 -5504.022} C_VEL
LIN {X 0,Y 509.241,Z 376.82,A -85,B 0,C 180,E1 -5504.078,E2 -5504.078} C_VEL
LIN {X 0,Y 509.284,Z 370.766,A -85,B 0,C 180,E1 -5506.846,E2 -5506.846} C_VEL
LIN {X 0,Y 509.451,Z 363.663,A -85,B 0,C 180,E1 -5510.174,E2 -5510.174} C_VEL
LIN {X 0,Y 509.481,Z 358.393,A -85,B 0,C 180,E1 -5512.721,E2 -5512.721} C_VEL
LIN {X 0,Y 509.585,Z 353.18,A -85,B 0,C 180,E1 -5515.311,E2 -5515.311} C_VEL
LIN {X 0,Y 509.736,Z 347.801,A -85,B 0,C 180,E1 -5518.066,E2 -5518.066} C_VEL
LIN {X 0,Y 509.898,Z 342.947,A -85,B 0,C 180,E1 -5520.662,E2 -5520.662} C_VEL
LIN {X 0,Y 510.069,Z 337.99,A -85,B 0,C 180,E1 -5523.445,E2 -5523.445} C_VEL
LIN {X 0,Y 510.235,Z 333.106,A -85,B 0,C 180,E1 -5526.319,E2 -5526.319} C_VEL
LIN {X 0,Y 510.415,Z 327.998,A -85,B 0,C 180,E1 -5529.549,E2 -5529.549} C_VEL
LIN {X 0,Y 510.476,Z 324.391,A -85,B 0,C 180,E1 -5531.974,E2 -5531.974} C_VEL
LIN {X 0,Y 510.227,Z 321.293,A -85,B 0,C 180,E1 -5534.253,E2 -5534.253} C_VEL
LIN {X 0,Y 509.824,Z 318.545,A -85,B 0,C 180,E1 -5536.428,E2 -5536.428} C_VEL
LIN {X 0,Y 509.839,Z 318.477,A -85,B 0,C 180,E1 -5539.302,E2 -5539.302} C_VEL
LIN {X 0,Y 509.852,Z 318.477,A -85,B 0,C 180,E1 -5541.786,E2 -5541.786} C_VEL
LIN {X 0,Y 509.83,Z 318.478,A -85,B 0,C 180,E1 -5544.622,E2 -5544.622} C_VEL
LIN {X 0,Y 509.862,Z 318.472,A -85,B 0,C 180,E1 -5547.48,E2 -5547.48} C_VEL
LIN {X 0,Y 509.859,Z 318.473,A -85,B 0,C 180,E1 -5550.273,E2 -5550.273} C_VEL
LIN {X 0,Y 509.884,Z 318.467,A -85,B 0,C 180,E1 -5552.944,E2 -5552.944} C_VEL
LIN {X 0,Y 509.851,Z 318.477,A -85,B 0,C 180,E1 -5555.573,E2 -5555.573} C_VEL
LIN {X 0,Y 509.822,Z 318.477,A -85,B 0,C 180,E1 -5558.148,E2 -5558.148} C_VEL
